//=============================================================================
// ST10_Flow5_FRobot_1.scl
// 1:1 CONVERSION FROM TIA PORTAL V18 GRAPH XML
// Generated: 2026-02-02
//=============================================================================

TYPE
    E_STEP_ST10_Flow5_FRobot_1 : (
        STEP_ST10_Flow5_FRobot_1_Tablecode_ScanFinish := 149,
        STEP_ST10_Flow5_FRobot_1_PickPalletProcess := 250,
        STEP_ST10_Flow5_FRobot_1_WaitRobotGripStatus := 360,
        STEP_ST10_Flow5_FRobot_1_WaitRobotFinish_4 := 356,
        STEP_ST10_Flow5_FRobot_1_WaitRobotFinish_9 := 371,
        STEP_ST10_Flow5_FRobot_1_WaitRobotGripStatus_4 := 372,
        STEP_ST10_Flow5_FRobot_1_WaitRobotGripHaveStatus_2 := 348,
        STEP_ST10_Flow5_FRobot_1_Open_NG_BOX_REQUESTED_ := 111,
        STEP_ST10_Flow5_FRobot_1_RobotReady_ := 311,
        STEP_ST10_Flow5_FRobot_1_WaitRobotGripStatus_6 := 378,
        STEP_ST10_Flow5_FRobot_1_Grip1SensorError := 379,
        STEP_ST10_Flow5_FRobot_1_ScanRing := 135,
        STEP_ST10_Flow5_FRobot_1_RobotAutoCycle := 329,
        STEP_ST10_Flow5_FRobot_1_RobotTaskSelect := 333,
        STEP_ST10_Flow5_FRobot_1_WaitRobotFinish_11 := 377,
        STEP_ST10_Flow5_FRobot_1_PartOKStatus_1 := 266,
        STEP_ST10_Flow5_FRobot_1_WaitRobotReachPos4 := 318,
        STEP_ST10_Flow5_FRobot_1_Step930 := 930,
        STEP_ST10_Flow5_FRobot_1_WaitR1MaintenPosFinsh := 702,
        STEP_ST10_Flow5_FRobot_1_WaitRobotGripStatus_3 := 369,
        STEP_ST10_Flow5_FRobot_1_WaitBrakeTestFinish := 921,
        STEP_ST10_Flow5_FRobot_1_PartOKStatus := 249,
        STEP_ST10_Flow5_FRobot_1_WaitGripperPos3ScanFinish := 340,
        STEP_ST10_Flow5_FRobot_1_DataMove_2 := 257,
        STEP_ST10_Flow5_FRobot_1_PressPick := 150,
        STEP_ST10_Flow5_FRobot_1_GripStatusCheck := 330,
        STEP_ST10_Flow5_FRobot_1_DataMove_5 := 264,
        STEP_ST10_Flow5_FRobot_1_NG2_PutProcessFinish := 799,
        STEP_ST10_Flow5_FRobot_1_WaitRobotReachPos5 := 321,
        STEP_ST10_Flow5_FRobot_1_StartRobotGluePut := 367,
        STEP_ST10_Flow5_FRobot_1_NG1Put_1_Press := 160,
        STEP_ST10_Flow5_FRobot_1_F5_Initial := 1,
        STEP_ST10_Flow5_FRobot_1_BrakeTestFinish := 929,
        STEP_ST10_Flow5_FRobot_1_StartRobotNG2Put_1 := 373,
        STEP_ST10_Flow5_FRobot_1_WaitPos4ScanFinish := 319,
        STEP_ST10_Flow5_FRobot_1_WaitRobotFinish := 327,
        STEP_ST10_Flow5_FRobot_1_WaitR1HomePosFinsh_1 := 899,
        STEP_ST10_Flow5_FRobot_1_NG1Put_2_ShaftScan := 165,
        STEP_ST10_Flow5_FRobot_1_FlagReset := 383,
        STEP_ST10_Flow5_FRobot_1_PressRingPutProcessFinish := 599,
        STEP_ST10_Flow5_FRobot_1_StartRobotNG3Put := 376,
        STEP_ST10_Flow5_FRobot_1_ScanStart := 246,
        STEP_ST10_Flow5_FRobot_1_StartRobotPutBuffer := 328,
        STEP_ST10_Flow5_FRobot_1_WaitMasteringTestFinish := 911,
        STEP_ST10_Flow5_FRobot_1_WaitRobotStartHome := 381,
        STEP_ST10_Flow5_FRobot_1_WaitScanCompletely := 247,
        STEP_ST10_Flow5_FRobot_1_DataMove_4 := 262,
        STEP_ST10_Flow5_FRobot_1_Grip1PartStatus := 243,
        STEP_ST10_Flow5_FRobot_1_StartRobotScanGripperCode := 334,
        STEP_ST10_Flow5_FRobot_1_WaitRobotFinish_5 := 359,
        STEP_ST10_Flow5_FRobot_1_WaitRobotGripHaveStatus := 346,
        STEP_ST10_Flow5_FRobot_1_WaitRobotFinish_1 := 343,
        STEP_ST10_Flow5_FRobot_1_WaitGripperPos1ScanFinish := 336,
        STEP_ST10_Flow5_FRobot_1_RobotStart := 316,
        STEP_ST10_Flow5_FRobot_1_WaitRobotReachPos2 := 313,
        STEP_ST10_Flow5_FRobot_1_PressShaftPut := 140,
        STEP_ST10_Flow5_FRobot_1_RobotHome := 317,
        STEP_ST10_Flow5_FRobot_1_WaitGripperPos4ScanFinish := 342,
        STEP_ST10_Flow5_FRobot_1_WaitRobotFinish_3 := 353,
        STEP_ST10_Flow5_FRobot_1_WaitRobotGripStatus_1 := 363,
        STEP_ST10_Flow5_FRobot_1_WaitPos2ScanFinish := 312,
        STEP_ST10_Flow5_FRobot_1_S10_InitialFinish := 10,
        STEP_ST10_Flow5_FRobot_1_PutBufferFinish_1 := 349,
        STEP_ST10_Flow5_FRobot_1_WaitRobotFinish_6 := 362,
        STEP_ST10_Flow5_FRobot_1_RobotScanGripperReachPos2 := 337,
        STEP_ST10_Flow5_FRobot_1_Grip2PartStatus := 244,
        STEP_ST10_Flow5_FRobot_1_WaitRobotGripStatus_2 := 366,
        STEP_ST10_Flow5_FRobot_1_WaitRobotReachPos6 := 322,
        STEP_ST10_Flow5_FRobot_1_RobotSpeed := 4,
        STEP_ST10_Flow5_FRobot_1_RobotTest := 900,
        STEP_ST10_Flow5_FRobot_1_WaitRobotHomeRequest := 703,
        STEP_ST10_Flow5_FRobot_1_PutBuffer := 120,
        STEP_ST10_Flow5_FRobot_1_StartRobotPickTable := 352,
        STEP_ST10_Flow5_FRobot_1_PickBufferFinish := 399,
        STEP_ST10_Flow5_FRobot_1_RobotScanGripperReachPos3 := 339,
        STEP_ST10_Flow5_FRobot_1_Grip2SensorError := 380,
        STEP_ST10_Flow5_FRobot_1_StartRobotPressPick := 364,
        STEP_ST10_Flow5_FRobot_1_ScanRingProcess := 450,
        STEP_ST10_Flow5_FRobot_1_GluePutProcess := 650,
        STEP_ST10_Flow5_FRobot_1_NG_2_PutProcess := 750,
        STEP_ST10_Flow5_FRobot_1_StartRobotNGPut := 370,
        STEP_ST10_Flow5_FRobot_1_Data_Clear_2 := 258,
        STEP_ST10_Flow5_FRobot_1_DataClear := 252,
        STEP_ST10_Flow5_FRobot_1_PressPickProcessFinish_ := 649,
        STEP_ST10_Flow5_FRobot_1_PickBuffer := 125,
        STEP_ST10_Flow5_FRobot_1_PickTableProcessFinish := 449,
        STEP_ST10_Flow5_FRobot_1_PressRingPutProcess := 550,
        STEP_ST10_Flow5_FRobot_1_NG_PutProcess := 700,
        STEP_ST10_Flow5_FRobot_1_WaitRobotFinish_2 := 345,
        STEP_ST10_Flow5_FRobot_1_PressRingPut := 145,
        STEP_ST10_Flow5_FRobot_1_WaitRobotGripHaveStatus_3 := 354,
        STEP_ST10_Flow5_FRobot_1_PickTableProcess := 400,
        STEP_ST10_Flow5_FRobot_1_WaitRobotReachPos3 := 314,
        STEP_ST10_Flow5_FRobot_1_Maintenance_Pos := 850,
        STEP_ST10_Flow5_FRobot_1_PressPickProcess := 600,
        STEP_ST10_Flow5_FRobot_1_Data_Clear_9 := 269,
        STEP_ST10_Flow5_FRobot_1_ProcessStart := 100,
        STEP_ST10_Flow5_FRobot_1_WaitGripperPos2ScanFinish := 338,
        STEP_ST10_Flow5_FRobot_1_Gripe2StatusAlarm := 332,
        STEP_ST10_Flow5_FRobot_1_MasteringTest_Req := 910,
        STEP_ST10_Flow5_FRobot_1_Tablecode_Scan := 200,
        STEP_ST10_Flow5_FRobot_1_Data_Clear_8 := 268,
        STEP_ST10_Flow5_FRobot_1_MES_Online__offline_ := 384,
        STEP_ST10_Flow5_FRobot_1_PartNGStatus := 251,
        STEP_ST10_Flow5_FRobot_1_S5_MESInitial := 5,
        STEP_ST10_Flow5_FRobot_1_StartRobotScanFixtureCode := 308,
        STEP_ST10_Flow5_FRobot_1_BrakeTest_Req := 920,
        STEP_ST10_Flow5_FRobot_1_WaitPos5ScanFinish := 320,
        STEP_ST10_Flow5_FRobot_1_RobotScanGripperReachPos4 := 341,
        STEP_ST10_Flow5_FRobot_1_ScanRingProcessFinish := 499,
        STEP_ST10_Flow5_FRobot_1_WaitRobotGripStatus_5 := 375,
        STEP_ST10_Flow5_FRobot_1_Masref_test := 132,
        STEP_ST10_Flow5_FRobot_1_WaitPos1ScanFinish := 310,
        STEP_ST10_Flow5_FRobot_1_StartRobotPressShaftPut := 358,
        STEP_ST10_Flow5_FRobot_1_StartRobotPickBuffer := 344,
        STEP_ST10_Flow5_FRobot_1_PressShaftPutProcess := 500,
        STEP_ST10_Flow5_FRobot_1_StartRobotPressRingPut := 361,
        STEP_ST10_Flow5_FRobot_1_NG1Put_3_RingScan := 170,
        STEP_ST10_Flow5_FRobot_1_NG1_PutProcessFinish := 749,
        STEP_ST10_Flow5_FRobot_1_WaitRobotReachScanPos := 357,
        STEP_ST10_Flow5_FRobot_1_PickPallet := 115,
        STEP_ST10_Flow5_FRobot_1_ScanFixtureCode := 110,
        STEP_ST10_Flow5_FRobot_1_PutBufferProcess := 300,
        STEP_ST10_Flow5_FRobot_1_WaitRobotFinish_10 := 374,
        STEP_ST10_Flow5_FRobot_1_ReqRobotToHomePos := 704,
        STEP_ST10_Flow5_FRobot_1_DataMove_1 := 255,
        STEP_ST10_Flow5_FRobot_1_Maintenance := 131,
        STEP_ST10_Flow5_FRobot_1_GluePut := 155,
        STEP_ST10_Flow5_FRobot_1_PickBufferProcess := 350,
        STEP_ST10_Flow5_FRobot_1_GluePutProcessFinish := 699,
        STEP_ST10_Flow5_FRobot_1_PickPalletFinish := 299,
        STEP_ST10_Flow5_FRobot_1_DataMove := 253,
        STEP_ST10_Flow5_FRobot_1_PressShaftPutProcessFinish := 549,
        STEP_ST10_Flow5_FRobot_1_StartRobotScanRing := 355,
        STEP_ST10_Flow5_FRobot_1_RobotManuallyMoved_ := 382,
        STEP_ST10_Flow5_FRobot_1_RobotScanGripperReachPos1 := 335,
        STEP_ST10_Flow5_FRobot_1_Data_Clear_7 := 267,
        STEP_ST10_Flow5_FRobot_1_CheckScanReady := 245,
        STEP_ST10_Flow5_FRobot_1_Brake_Test := 133,
        STEP_ST10_Flow5_FRobot_1_ReqRobotToMantenPos := 701,
        STEP_ST10_Flow5_FRobot_1_NG3_PutProcessFinish := 849,
        STEP_ST10_Flow5_FRobot_1_NG_3_PutProcess := 800,
        STEP_ST10_Flow5_FRobot_1_Wait_ScanFinish := 242,
        STEP_ST10_Flow5_FRobot_1_WaitRobotReachPos1 := 309,
        STEP_ST10_Flow5_FRobot_1_WaitRobotGripHaveStatus_1 := 347,
        STEP_ST10_Flow5_FRobot_1_DataMove_3 := 260,
        STEP_ST10_Flow5_FRobot_1_MasteringTestFinish := 919,
        STEP_ST10_Flow5_FRobot_1_StartRobotPickPalletShaft := 326,
        STEP_ST10_Flow5_FRobot_1_PickTable := 130,
        STEP_ST10_Flow5_FRobot_1_WaitRobotFinish_8 := 368,
        STEP_ST10_Flow5_FRobot_1_Gripe1StatusAlarm := 331,
        STEP_ST10_Flow5_FRobot_1_CodeMove := 248,
        STEP_ST10_Flow5_FRobot_1_WaitPos3ScanFinish := 315,
        STEP_ST10_Flow5_FRobot_1_WaitRobotFinish_7 := 365,
    ) INT := 1;
END_TYPE

CONST
    STEP_ST10_Flow5_FRobot_1_Tablecode_ScanFinish := 149;
    STEP_ST10_Flow5_FRobot_1_PickPalletProcess := 250;
    STEP_ST10_Flow5_FRobot_1_WaitRobotGripStatus := 360;
    STEP_ST10_Flow5_FRobot_1_WaitRobotFinish_4 := 356;
    STEP_ST10_Flow5_FRobot_1_WaitRobotFinish_9 := 371;
    STEP_ST10_Flow5_FRobot_1_WaitRobotGripStatus_4 := 372;
    STEP_ST10_Flow5_FRobot_1_WaitRobotGripHaveStatus_2 := 348;
    STEP_ST10_Flow5_FRobot_1_Open_NG_BOX_REQUESTED_ := 111;
    STEP_ST10_Flow5_FRobot_1_RobotReady_ := 311;
    STEP_ST10_Flow5_FRobot_1_WaitRobotGripStatus_6 := 378;
    STEP_ST10_Flow5_FRobot_1_Grip1SensorError := 379;
    STEP_ST10_Flow5_FRobot_1_ScanRing := 135;
    STEP_ST10_Flow5_FRobot_1_RobotAutoCycle := 329;
    STEP_ST10_Flow5_FRobot_1_RobotTaskSelect := 333;
    STEP_ST10_Flow5_FRobot_1_WaitRobotFinish_11 := 377;
    STEP_ST10_Flow5_FRobot_1_PartOKStatus_1 := 266;
    STEP_ST10_Flow5_FRobot_1_WaitRobotReachPos4 := 318;
    STEP_ST10_Flow5_FRobot_1_Step930 := 930;
    STEP_ST10_Flow5_FRobot_1_WaitR1MaintenPosFinsh := 702;
    STEP_ST10_Flow5_FRobot_1_WaitRobotGripStatus_3 := 369;
    STEP_ST10_Flow5_FRobot_1_WaitBrakeTestFinish := 921;
    STEP_ST10_Flow5_FRobot_1_PartOKStatus := 249;
    STEP_ST10_Flow5_FRobot_1_WaitGripperPos3ScanFinish := 340;
    STEP_ST10_Flow5_FRobot_1_DataMove_2 := 257;
    STEP_ST10_Flow5_FRobot_1_PressPick := 150;
    STEP_ST10_Flow5_FRobot_1_GripStatusCheck := 330;
    STEP_ST10_Flow5_FRobot_1_DataMove_5 := 264;
    STEP_ST10_Flow5_FRobot_1_NG2_PutProcessFinish := 799;
    STEP_ST10_Flow5_FRobot_1_WaitRobotReachPos5 := 321;
    STEP_ST10_Flow5_FRobot_1_StartRobotGluePut := 367;
    STEP_ST10_Flow5_FRobot_1_NG1Put_1_Press := 160;
    STEP_ST10_Flow5_FRobot_1_F5_Initial := 1;
    STEP_ST10_Flow5_FRobot_1_BrakeTestFinish := 929;
    STEP_ST10_Flow5_FRobot_1_StartRobotNG2Put_1 := 373;
    STEP_ST10_Flow5_FRobot_1_WaitPos4ScanFinish := 319;
    STEP_ST10_Flow5_FRobot_1_WaitRobotFinish := 327;
    STEP_ST10_Flow5_FRobot_1_WaitR1HomePosFinsh_1 := 899;
    STEP_ST10_Flow5_FRobot_1_NG1Put_2_ShaftScan := 165;
    STEP_ST10_Flow5_FRobot_1_FlagReset := 383;
    STEP_ST10_Flow5_FRobot_1_PressRingPutProcessFinish := 599;
    STEP_ST10_Flow5_FRobot_1_StartRobotNG3Put := 376;
    STEP_ST10_Flow5_FRobot_1_ScanStart := 246;
    STEP_ST10_Flow5_FRobot_1_StartRobotPutBuffer := 328;
    STEP_ST10_Flow5_FRobot_1_WaitMasteringTestFinish := 911;
    STEP_ST10_Flow5_FRobot_1_WaitRobotStartHome := 381;
    STEP_ST10_Flow5_FRobot_1_WaitScanCompletely := 247;
    STEP_ST10_Flow5_FRobot_1_DataMove_4 := 262;
    STEP_ST10_Flow5_FRobot_1_Grip1PartStatus := 243;
    STEP_ST10_Flow5_FRobot_1_StartRobotScanGripperCode := 334;
    STEP_ST10_Flow5_FRobot_1_WaitRobotFinish_5 := 359;
    STEP_ST10_Flow5_FRobot_1_WaitRobotGripHaveStatus := 346;
    STEP_ST10_Flow5_FRobot_1_WaitRobotFinish_1 := 343;
    STEP_ST10_Flow5_FRobot_1_WaitGripperPos1ScanFinish := 336;
    STEP_ST10_Flow5_FRobot_1_RobotStart := 316;
    STEP_ST10_Flow5_FRobot_1_WaitRobotReachPos2 := 313;
    STEP_ST10_Flow5_FRobot_1_PressShaftPut := 140;
    STEP_ST10_Flow5_FRobot_1_RobotHome := 317;
    STEP_ST10_Flow5_FRobot_1_WaitGripperPos4ScanFinish := 342;
    STEP_ST10_Flow5_FRobot_1_WaitRobotFinish_3 := 353;
    STEP_ST10_Flow5_FRobot_1_WaitRobotGripStatus_1 := 363;
    STEP_ST10_Flow5_FRobot_1_WaitPos2ScanFinish := 312;
    STEP_ST10_Flow5_FRobot_1_S10_InitialFinish := 10;
    STEP_ST10_Flow5_FRobot_1_PutBufferFinish_1 := 349;
    STEP_ST10_Flow5_FRobot_1_WaitRobotFinish_6 := 362;
    STEP_ST10_Flow5_FRobot_1_RobotScanGripperReachPos2 := 337;
    STEP_ST10_Flow5_FRobot_1_Grip2PartStatus := 244;
    STEP_ST10_Flow5_FRobot_1_WaitRobotGripStatus_2 := 366;
    STEP_ST10_Flow5_FRobot_1_WaitRobotReachPos6 := 322;
    STEP_ST10_Flow5_FRobot_1_RobotSpeed := 4;
    STEP_ST10_Flow5_FRobot_1_RobotTest := 900;
    STEP_ST10_Flow5_FRobot_1_WaitRobotHomeRequest := 703;
    STEP_ST10_Flow5_FRobot_1_PutBuffer := 120;
    STEP_ST10_Flow5_FRobot_1_StartRobotPickTable := 352;
    STEP_ST10_Flow5_FRobot_1_PickBufferFinish := 399;
    STEP_ST10_Flow5_FRobot_1_RobotScanGripperReachPos3 := 339;
    STEP_ST10_Flow5_FRobot_1_Grip2SensorError := 380;
    STEP_ST10_Flow5_FRobot_1_StartRobotPressPick := 364;
    STEP_ST10_Flow5_FRobot_1_ScanRingProcess := 450;
    STEP_ST10_Flow5_FRobot_1_GluePutProcess := 650;
    STEP_ST10_Flow5_FRobot_1_NG_2_PutProcess := 750;
    STEP_ST10_Flow5_FRobot_1_StartRobotNGPut := 370;
    STEP_ST10_Flow5_FRobot_1_Data_Clear_2 := 258;
    STEP_ST10_Flow5_FRobot_1_DataClear := 252;
    STEP_ST10_Flow5_FRobot_1_PressPickProcessFinish_ := 649;
    STEP_ST10_Flow5_FRobot_1_PickBuffer := 125;
    STEP_ST10_Flow5_FRobot_1_PickTableProcessFinish := 449;
    STEP_ST10_Flow5_FRobot_1_PressRingPutProcess := 550;
    STEP_ST10_Flow5_FRobot_1_NG_PutProcess := 700;
    STEP_ST10_Flow5_FRobot_1_WaitRobotFinish_2 := 345;
    STEP_ST10_Flow5_FRobot_1_PressRingPut := 145;
    STEP_ST10_Flow5_FRobot_1_WaitRobotGripHaveStatus_3 := 354;
    STEP_ST10_Flow5_FRobot_1_PickTableProcess := 400;
    STEP_ST10_Flow5_FRobot_1_WaitRobotReachPos3 := 314;
    STEP_ST10_Flow5_FRobot_1_Maintenance_Pos := 850;
    STEP_ST10_Flow5_FRobot_1_PressPickProcess := 600;
    STEP_ST10_Flow5_FRobot_1_Data_Clear_9 := 269;
    STEP_ST10_Flow5_FRobot_1_ProcessStart := 100;
    STEP_ST10_Flow5_FRobot_1_WaitGripperPos2ScanFinish := 338;
    STEP_ST10_Flow5_FRobot_1_Gripe2StatusAlarm := 332;
    STEP_ST10_Flow5_FRobot_1_MasteringTest_Req := 910;
    STEP_ST10_Flow5_FRobot_1_Tablecode_Scan := 200;
    STEP_ST10_Flow5_FRobot_1_Data_Clear_8 := 268;
    STEP_ST10_Flow5_FRobot_1_MES_Online__offline_ := 384;
    STEP_ST10_Flow5_FRobot_1_PartNGStatus := 251;
    STEP_ST10_Flow5_FRobot_1_S5_MESInitial := 5;
    STEP_ST10_Flow5_FRobot_1_StartRobotScanFixtureCode := 308;
    STEP_ST10_Flow5_FRobot_1_BrakeTest_Req := 920;
    STEP_ST10_Flow5_FRobot_1_WaitPos5ScanFinish := 320;
    STEP_ST10_Flow5_FRobot_1_RobotScanGripperReachPos4 := 341;
    STEP_ST10_Flow5_FRobot_1_ScanRingProcessFinish := 499;
    STEP_ST10_Flow5_FRobot_1_WaitRobotGripStatus_5 := 375;
    STEP_ST10_Flow5_FRobot_1_Masref_test := 132;
    STEP_ST10_Flow5_FRobot_1_WaitPos1ScanFinish := 310;
    STEP_ST10_Flow5_FRobot_1_StartRobotPressShaftPut := 358;
    STEP_ST10_Flow5_FRobot_1_StartRobotPickBuffer := 344;
    STEP_ST10_Flow5_FRobot_1_PressShaftPutProcess := 500;
    STEP_ST10_Flow5_FRobot_1_StartRobotPressRingPut := 361;
    STEP_ST10_Flow5_FRobot_1_NG1Put_3_RingScan := 170;
    STEP_ST10_Flow5_FRobot_1_NG1_PutProcessFinish := 749;
    STEP_ST10_Flow5_FRobot_1_WaitRobotReachScanPos := 357;
    STEP_ST10_Flow5_FRobot_1_PickPallet := 115;
    STEP_ST10_Flow5_FRobot_1_ScanFixtureCode := 110;
    STEP_ST10_Flow5_FRobot_1_PutBufferProcess := 300;
    STEP_ST10_Flow5_FRobot_1_WaitRobotFinish_10 := 374;
    STEP_ST10_Flow5_FRobot_1_ReqRobotToHomePos := 704;
    STEP_ST10_Flow5_FRobot_1_DataMove_1 := 255;
    STEP_ST10_Flow5_FRobot_1_Maintenance := 131;
    STEP_ST10_Flow5_FRobot_1_GluePut := 155;
    STEP_ST10_Flow5_FRobot_1_PickBufferProcess := 350;
    STEP_ST10_Flow5_FRobot_1_GluePutProcessFinish := 699;
    STEP_ST10_Flow5_FRobot_1_PickPalletFinish := 299;
    STEP_ST10_Flow5_FRobot_1_DataMove := 253;
    STEP_ST10_Flow5_FRobot_1_PressShaftPutProcessFinish := 549;
    STEP_ST10_Flow5_FRobot_1_StartRobotScanRing := 355;
    STEP_ST10_Flow5_FRobot_1_RobotManuallyMoved_ := 382;
    STEP_ST10_Flow5_FRobot_1_RobotScanGripperReachPos1 := 335;
    STEP_ST10_Flow5_FRobot_1_Data_Clear_7 := 267;
    STEP_ST10_Flow5_FRobot_1_CheckScanReady := 245;
    STEP_ST10_Flow5_FRobot_1_Brake_Test := 133;
    STEP_ST10_Flow5_FRobot_1_ReqRobotToMantenPos := 701;
    STEP_ST10_Flow5_FRobot_1_NG3_PutProcessFinish := 849;
    STEP_ST10_Flow5_FRobot_1_NG_3_PutProcess := 800;
    STEP_ST10_Flow5_FRobot_1_Wait_ScanFinish := 242;
    STEP_ST10_Flow5_FRobot_1_WaitRobotReachPos1 := 309;
    STEP_ST10_Flow5_FRobot_1_WaitRobotGripHaveStatus_1 := 347;
    STEP_ST10_Flow5_FRobot_1_DataMove_3 := 260;
    STEP_ST10_Flow5_FRobot_1_MasteringTestFinish := 919;
    STEP_ST10_Flow5_FRobot_1_StartRobotPickPalletShaft := 326;
    STEP_ST10_Flow5_FRobot_1_PickTable := 130;
    STEP_ST10_Flow5_FRobot_1_WaitRobotFinish_8 := 368;
    STEP_ST10_Flow5_FRobot_1_Gripe1StatusAlarm := 331;
    STEP_ST10_Flow5_FRobot_1_CodeMove := 248;
    STEP_ST10_Flow5_FRobot_1_WaitPos3ScanFinish := 315;
    STEP_ST10_Flow5_FRobot_1_WaitRobotFinish_7 := 365;
END_CONST

FUNCTION_BLOCK "ST10_Flow5_FRobot_1_1to1"
{ S7_Optimized_Access := 'TRUE' }
VERSION : 1.0

VAR_INPUT
    iSysInface : "RCS_SysComInterface_V1";
END_VAR

VAR_IN_OUT
    ioPM_Inface : "RCS_PMInterface_V1";
    ioStatus : Int;
END_VAR

VAR_OUTPUT
    oAlarmID : Int;
END_VAR

VAR
    State : INT := 1;
    act_InitialRun : Bool;
    act_InitialOK : Bool;
    act_WaitRunning : Bool;
    act_Running : Bool;
    act_ProcessComplete : Bool;
    act_ProcessStart : Bool;
    act_UnPause : Bool;
    bError : Bool;
    wErrorID : Word;
END_VAR

BEGIN
    //======================================================================
    // STATE MACHINE - Inline Transition Conditions
    //======================================================================

    CASE #State OF

        // ===========================================
        // STEP 149: Tablecode ScanFinish
        // ===========================================
        STEP_ST10_Flow5_FRobot_1_Tablecode_ScanFinish:
            // Action Qualifier=S
            // Token: #ioPM_Inface.ProcessComplete
            #ioPM_Inface.ProcessComplete := TRUE;
            // Action Qualifier=R
            // Token: #ioPM_Inface.ProcessStart
            #ioPM_Inface.ProcessStart := FALSE;

            // Transition to next step: 250
            IF TRUE THEN  // Sequential transition - review XML for actual condition
                #State := STEP_ST10_Flow5_FRobot_1_PickPalletProcess;
            END_IF;

        // ===========================================
        // STEP 250: PickPalletProcess
        // ===========================================
        STEP_ST10_Flow5_FRobot_1_PickPalletProcess:
            // No actions in XML

            // Transition to next step: 360
            IF TRUE THEN  // Sequential transition - review XML for actual condition
                #State := STEP_ST10_Flow5_FRobot_1_WaitRobotGripStatus;
            END_IF;

        // ===========================================
        // STEP 360: WaitRobotGripStatus
        // ===========================================
        STEP_ST10_Flow5_FRobot_1_WaitRobotGripStatus:
            // No actions in XML

            // Transition to next step: 356
            IF TRUE THEN  // Sequential transition - review XML for actual condition
                #State := STEP_ST10_Flow5_FRobot_1_WaitRobotFinish_4;
            END_IF;

        // ===========================================
        // STEP 356: WaitRobotFinish_4
        // ===========================================
        STEP_ST10_Flow5_FRobot_1_WaitRobotFinish_4:
            // Action Qualifier=N
            // Token: "KukaRobot1_CtrlDB".sPLCtoROB.User.Cycle.DI262_RingScanComplete
            "KukaRobot1_CtrlDB".sPLCtoROB.User.Cycle.DI262_RingScanComplete;

            // Transition to next step: 371
            IF TRUE THEN  // Sequential transition - review XML for actual condition
                #State := STEP_ST10_Flow5_FRobot_1_WaitRobotFinish_9;
            END_IF;

        // ===========================================
        // STEP 371: WaitRobotFinish_9
        // ===========================================
        STEP_ST10_Flow5_FRobot_1_WaitRobotFinish_9:
            // No actions in XML

            // Transition to next step: 372
            IF TRUE THEN  // Sequential transition - review XML for actual condition
                #State := STEP_ST10_Flow5_FRobot_1_WaitRobotGripStatus_4;
            END_IF;

        // ===========================================
        // STEP 372: WaitRobotGripStatus_4
        // ===========================================
        STEP_ST10_Flow5_FRobot_1_WaitRobotGripStatus_4:
            // No actions in XML

            // Transition to next step: 348
            IF TRUE THEN  // Sequential transition - review XML for actual condition
                #State := STEP_ST10_Flow5_FRobot_1_WaitRobotGripHaveStatus_2;
            END_IF;

        // ===========================================
        // STEP 348: WaitRobotGripHaveStatus_2
        // ===========================================
        STEP_ST10_Flow5_FRobot_1_WaitRobotGripHaveStatus_2:
            // No actions in XML

            // Transition to next step: 111
            IF TRUE THEN  // Sequential transition - review XML for actual condition
                #State := STEP_ST10_Flow5_FRobot_1_Open_NG_BOX_REQUESTED_;
            END_IF;

        // ===========================================
        // STEP 111: Open NG BOX REQUESTED?
        // ===========================================
        STEP_ST10_Flow5_FRobot_1_Open_NG_BOX_REQUESTED_:
            // No actions in XML

            // Transition to next step: 311
            IF TRUE THEN  // Sequential transition - review XML for actual condition
                #State := STEP_ST10_Flow5_FRobot_1_RobotReady_;
            END_IF;

        // ===========================================
        // STEP 311: RobotReady?
        // ===========================================
        STEP_ST10_Flow5_FRobot_1_RobotReady_:
            // No actions in XML

            // Transition to next step: 378
            IF TRUE THEN  // Sequential transition - review XML for actual condition
                #State := STEP_ST10_Flow5_FRobot_1_WaitRobotGripStatus_6;
            END_IF;

        // ===========================================
        // STEP 378: WaitRobotGripStatus_6
        // ===========================================
        STEP_ST10_Flow5_FRobot_1_WaitRobotGripStatus_6:
            // No actions in XML

            // Transition to next step: 379
            IF TRUE THEN  // Sequential transition - review XML for actual condition
                #State := STEP_ST10_Flow5_FRobot_1_Grip1SensorError;
            END_IF;

        // ===========================================
        // STEP 379: Grip1SensorError
        // ===========================================
        STEP_ST10_Flow5_FRobot_1_Grip1SensorError:
            // No actions in XML

            // Transition to next step: 135
            IF TRUE THEN  // Sequential transition - review XML for actual condition
                #State := STEP_ST10_Flow5_FRobot_1_ScanRing;
            END_IF;

        // ===========================================
        // STEP 135: ScanRing
        // ===========================================
        STEP_ST10_Flow5_FRobot_1_ScanRing:
            // Action Qualifier=R
            // Token: #ioPM_Inface.ProcessComplete
            #ioPM_Inface.ProcessComplete := FALSE;
            // Action Qualifier=S
            // Token: #ioPM_Inface.ProcessStart
            #ioPM_Inface.ProcessStart := TRUE;

            // Transition to next step: 329
            IF TRUE THEN  // Sequential transition - review XML for actual condition
                #State := STEP_ST10_Flow5_FRobot_1_RobotAutoCycle;
            END_IF;

        // ===========================================
        // STEP 329: RobotAutoCycle
        // ===========================================
        STEP_ST10_Flow5_FRobot_1_RobotAutoCycle:
            // Action Qualifier=N
            // Token: "KukaRobot1_CtrlDB".ioStartAutoCycle
            "KukaRobot1_CtrlDB".ioStartAutoCycle;

            // Transition to next step: 333
            IF TRUE THEN  // Sequential transition - review XML for actual condition
                #State := STEP_ST10_Flow5_FRobot_1_RobotTaskSelect;
            END_IF;

        // ===========================================
        // STEP 333: RobotTaskSelect
        // ===========================================
        STEP_ST10_Flow5_FRobot_1_RobotTaskSelect:
            // No actions in XML

            // Transition to next step: 377
            IF TRUE THEN  // Sequential transition - review XML for actual condition
                #State := STEP_ST10_Flow5_FRobot_1_WaitRobotFinish_11;
            END_IF;

        // ===========================================
        // STEP 377: WaitRobotFinish_11
        // ===========================================
        STEP_ST10_Flow5_FRobot_1_WaitRobotFinish_11:
            // No actions in XML

            // Transition to next step: 266
            IF TRUE THEN  // Sequential transition - review XML for actual condition
                #State := STEP_ST10_Flow5_FRobot_1_PartOKStatus_1;
            END_IF;

        // ===========================================
        // STEP 266: PartOKStatus_1
        // ===========================================
        STEP_ST10_Flow5_FRobot_1_PartOKStatus_1:
            // Action Qualifier=N
            // Token: "AutoProcessData".F_Robot1Grip2.PartStatus := 110
            "AutoProcessData".F_Robot1Grip2.PartStatus := 110;

            // Transition to next step: 318
            IF TRUE THEN  // Sequential transition - review XML for actual condition
                #State := STEP_ST10_Flow5_FRobot_1_WaitRobotReachPos4;
            END_IF;

        // ===========================================
        // STEP 318: WaitRobotReachPos4
        // ===========================================
        STEP_ST10_Flow5_FRobot_1_WaitRobotReachPos4:
            // No actions in XML

            // Transition to next step: 930
            IF TRUE THEN  // Sequential transition - review XML for actual condition
                #State := STEP_ST10_Flow5_FRobot_1_Step930;
            END_IF;

        // ===========================================
        // STEP 930: Step930
        // ===========================================
        STEP_ST10_Flow5_FRobot_1_Step930:
            // No actions in XML

            // Transition to next step: 702
            IF TRUE THEN  // Sequential transition - review XML for actual condition
                #State := STEP_ST10_Flow5_FRobot_1_WaitR1MaintenPosFinsh;
            END_IF;

        // ===========================================
        // STEP 702: WaitR1MaintenPosFinsh
        // ===========================================
        STEP_ST10_Flow5_FRobot_1_WaitR1MaintenPosFinsh:
            // Action Qualifier=R
            // Token: "AutoProcessControl".Robot_1.MaintenanceRequest
            "AutoProcessControl".Robot_1.MaintenanceRequest := FALSE;

            // Transition to next step: 369
            IF TRUE THEN  // Sequential transition - review XML for actual condition
                #State := STEP_ST10_Flow5_FRobot_1_WaitRobotGripStatus_3;
            END_IF;

        // ===========================================
        // STEP 369: WaitRobotGripStatus_3
        // ===========================================
        STEP_ST10_Flow5_FRobot_1_WaitRobotGripStatus_3:
            // No actions in XML

            // Transition to next step: 921
            IF TRUE THEN  // Sequential transition - review XML for actual condition
                #State := STEP_ST10_Flow5_FRobot_1_WaitBrakeTestFinish;
            END_IF;

        // ===========================================
        // STEP 921: WaitBrakeTestFinish
        // ===========================================
        STEP_ST10_Flow5_FRobot_1_WaitBrakeTestFinish:
            // No actions in XML

            // Transition to next step: 249
            IF TRUE THEN  // Sequential transition - review XML for actual condition
                #State := STEP_ST10_Flow5_FRobot_1_PartOKStatus;
            END_IF;

        // ===========================================
        // STEP 249: PartOKStatus
        // ===========================================
        STEP_ST10_Flow5_FRobot_1_PartOKStatus:
            // Action Qualifier=N
            // Token: "AutoProcessData".F_Robot1Grip2.PartStatus := 199
            "AutoProcessData".F_Robot1Grip2.PartStatus := 199;

            // Transition to next step: 340
            IF TRUE THEN  // Sequential transition - review XML for actual condition
                #State := STEP_ST10_Flow5_FRobot_1_WaitGripperPos3ScanFinish;
            END_IF;

        // ===========================================
        // STEP 340: WaitGripperPos3ScanFinish
        // ===========================================
        STEP_ST10_Flow5_FRobot_1_WaitGripperPos3ScanFinish:
            // No actions in XML

            // Transition to next step: 257
            IF TRUE THEN  // Sequential transition - review XML for actual condition
                #State := STEP_ST10_Flow5_FRobot_1_DataMove_2;
            END_IF;

        // ===========================================
        // STEP 257: DataMove_2
        // ===========================================
        STEP_ST10_Flow5_FRobot_1_DataMove_2:
            // Action Qualifier=N, Event="S1"
            // Token: "AutoProcessData".B_Press1 := "AutoProcessData".F_Robot1Grip1
            "AutoProcessData".B_Press1 := "AutoProcessData".F_Robot1Grip1;
            // Action Qualifier=N, Event="S1"
            // Token: "AutoProcessData".F_Robot1Grip1 := "AutoProcessData".ClearData
            "AutoProcessData".F_Robot1Grip1 := "AutoProcessData".ClearData;

            // Transition to next step: 150
            IF TRUE THEN  // Sequential transition - review XML for actual condition
                #State := STEP_ST10_Flow5_FRobot_1_PressPick;
            END_IF;

        // ===========================================
        // STEP 150: PressPick
        // ===========================================
        STEP_ST10_Flow5_FRobot_1_PressPick:
            // Action Qualifier=R
            // Token: #ioPM_Inface.ProcessComplete
            #ioPM_Inface.ProcessComplete := FALSE;
            // Action Qualifier=S
            // Token: #ioPM_Inface.ProcessStart
            #ioPM_Inface.ProcessStart := TRUE;

            // Transition to next step: 330
            IF TRUE THEN  // Sequential transition - review XML for actual condition
                #State := STEP_ST10_Flow5_FRobot_1_GripStatusCheck;
            END_IF;

        // ===========================================
        // STEP 330: GripStatusCheck
        // ===========================================
        STEP_ST10_Flow5_FRobot_1_GripStatusCheck:
            // No actions in XML

            // Transition to next step: 264
            IF TRUE THEN  // Sequential transition - review XML for actual condition
                #State := STEP_ST10_Flow5_FRobot_1_DataMove_5;
            END_IF;

        // ===========================================
        // STEP 264: DataMove_5
        // ===========================================
        STEP_ST10_Flow5_FRobot_1_DataMove_5:
            // Action Qualifier=N, Event="S1"
            // Token: "AutoProcessData".C_Glue := "AutoProcessData".F_Robot1Grip1
            "AutoProcessData".C_Glue := "AutoProcessData".F_Robot1Grip1;
            // Action Qualifier=N, Event="S1"
            // Token: "AutoProcessData".F_Robot1Grip1 := "AutoProcessData".ClearData
            "AutoProcessData".F_Robot1Grip1 := "AutoProcessData".ClearData;

            // Transition to next step: 799
            IF TRUE THEN  // Sequential transition - review XML for actual condition
                #State := STEP_ST10_Flow5_FRobot_1_NG2_PutProcessFinish;
            END_IF;

        // ===========================================
        // STEP 799: NG2 PutProcessFinish
        // ===========================================
        STEP_ST10_Flow5_FRobot_1_NG2_PutProcessFinish:
            // Action Qualifier=S
            // Token: #ioPM_Inface.ProcessComplete
            #ioPM_Inface.ProcessComplete := TRUE;
            // Action Qualifier=R
            // Token: #ioPM_Inface.ProcessStart
            #ioPM_Inface.ProcessStart := FALSE;

            // Transition to next step: 321
            IF TRUE THEN  // Sequential transition - review XML for actual condition
                #State := STEP_ST10_Flow5_FRobot_1_WaitRobotReachPos5;
            END_IF;

        // ===========================================
        // STEP 321: WaitRobotReachPos5
        // ===========================================
        STEP_ST10_Flow5_FRobot_1_WaitRobotReachPos5:
            // No actions in XML

            // Transition to next step: 367
            IF TRUE THEN  // Sequential transition - review XML for actual condition
                #State := STEP_ST10_Flow5_FRobot_1_StartRobotGluePut;
            END_IF;

        // ===========================================
        // STEP 367: StartRobotGluePut
        // ===========================================
        STEP_ST10_Flow5_FRobot_1_StartRobotGluePut:
            // Action Qualifier=N
            // Token: "KukaRobot1_CtrlDB".sPLCtoROB.User.Cycle.DI289_GluePutReq
            "KukaRobot1_CtrlDB".sPLCtoROB.User.Cycle.DI289_GluePutReq;

            // Transition to next step: 160
            IF TRUE THEN  // Sequential transition - review XML for actual condition
                #State := STEP_ST10_Flow5_FRobot_1_NG1Put_1_Press;
            END_IF;

        // ===========================================
        // STEP 160: NG1Put_1/Press
        // ===========================================
        STEP_ST10_Flow5_FRobot_1_NG1Put_1_Press:
            // Action Qualifier=S
            // Token: "AutoProcessControl".Robot_1.NGPutFlag
            "AutoProcessControl".Robot_1.NGPutFlag := TRUE;
            // Action Qualifier=R
            // Token: #ioPM_Inface.ProcessComplete
            #ioPM_Inface.ProcessComplete := FALSE;
            // Action Qualifier=S
            // Token: #ioPM_Inface.ProcessStart
            #ioPM_Inface.ProcessStart := TRUE;

            // Transition to next step: 1
            IF TRUE THEN  // Sequential transition - review XML for actual condition
                #State := STEP_ST10_Flow5_FRobot_1_F5_Initial;
            END_IF;

        // ===========================================
        // STEP 1: F5_Initial
        // ===========================================
        STEP_ST10_Flow5_FRobot_1_F5_Initial:
            // Action Qualifier=S
            // Token: #ioPM_Inface.InitialRun
            #ioPM_Inface.InitialRun := TRUE;
            // Action Qualifier=R
            // Token: #ioPM_Inface.InitialOK
            #ioPM_Inface.InitialOK := FALSE;
            // Action Qualifier=R
            // Token: #ioPM_Inface.WaitRunning
            #ioPM_Inface.WaitRunning := FALSE;
            // Action Qualifier=R
            // Token: #ioPM_Inface.Running
            #ioPM_Inface.Running := FALSE;
            // Action Qualifier=R
            // Token: #ioPM_Inface.UnPause
            #ioPM_Inface.UnPause := FALSE;
            // Action Qualifier=R
            // Token: "Station_Sys".Cmd.Calibration
            "Station_Sys".Cmd.Calibration := FALSE;
            // Action Qualifier=R
            // Token: "Station_Sys".Cmd.ChangeOver
            "Station_Sys".Cmd.ChangeOver := FALSE;
            // Action Qualifier=N
            // Token: //"ST350_Sys".Cmd.DryRun
            //"ST350_Sys".Cmd.DryRun;
            // Action Qualifier=R
            // Token: "Station_Sys".Cmd.Reserve
            "Station_Sys".Cmd.Reserve := FALSE;
            // Action Qualifier=R
            // Token: "Station_Sys".Cmd.OneCycle
            "Station_Sys".Cmd.OneCycle := FALSE;
            // Action Qualifier=R
            // Token: "AutoProcessControl".Robot_1.GluePutFlag
            "AutoProcessControl".Robot_1.GluePutFlag := FALSE;
            // Action Qualifier=R
            // Token: "AutoProcessControl".Robot_1.NGPutFlag
            "AutoProcessControl".Robot_1.NGPutFlag := FALSE;
            // Action Qualifier=R
            // Token: #ioPM_Inface.ProcessComplete
            #ioPM_Inface.ProcessComplete := FALSE;
            // Action Qualifier=R
            // Token: #ioPM_Inface.ProcessStart
            #ioPM_Inface.ProcessStart := FALSE;
            // Action Qualifier=R
            // Token: "ChangeOver_DB".Robot_1.MaintenancePosReqSelFlag
            "ChangeOver_DB".Robot_1.MaintenancePosReqSelFlag := FALSE;
            // Action Qualifier=N
            // Token: //"Robot_DB".Robot_1.MasteringTest_Req
            //"Robot_DB".Robot_1.MasteringTest_Req;
            // Action Qualifier=N
            // Token: //"Robot_DB".Robot_1.BrakeTest_Req
            //"Robot_DB".Robot_1.BrakeTest_Req;
            // Action Qualifier=R
            // Token: "KukaRobot1_CtrlDB".sPLCtoROB.User.Cycle.DI281_PressPickShaftReq
            "KukaRobot1_CtrlDB".sPLCtoROB.User.Cycle.DI281_PressPickShaftReq := FALSE;
            // Action Qualifier=R
            // Token: "KukaRobot1_CtrlDB".sPLCtoROB.User.Cycle.DI277_PressRingPutReq
            "KukaRobot1_CtrlDB".sPLCtoROB.User.Cycle.DI277_PressRingPutReq := FALSE;
            // Action Qualifier=R
            // Token: "KukaRobot1_CtrlDB".sPLCtoROB.User.Cycle.DI278_PressRingPutLeave
            "KukaRobot1_CtrlDB".sPLCtoROB.User.Cycle.DI278_PressRingPutLeave := FALSE;
            // Action Qualifier=R
            // Token: "KukaRobot1_CtrlDB".sPLCtoROB.User.Cycle.DI267_LoadRingScanNGReq3
            "KukaRobot1_CtrlDB".sPLCtoROB.User.Cycle.DI267_LoadRingScanNGReq3 := FALSE;
            // Action Qualifier=R
            // Token: "KukaRobot1_CtrlDB".sPLCtoROB.User.Cycle.DI265_LoadPressNGReq1
            "KukaRobot1_CtrlDB".sPLCtoROB.User.Cycle.DI265_LoadPressNGReq1 := FALSE;
            // Action Qualifier=R
            // Token: "KukaRobot1_CtrlDB".sPLCtoROB.User.Cycle.DI261_RingScanReq
            "KukaRobot1_CtrlDB".sPLCtoROB.User.Cycle.DI261_RingScanReq := FALSE;
            // Action Qualifier=R
            // Token: "KukaRobot1_CtrlDB".sPLCtoROB.User.Cycle.DI262_RingScanComplete
            "KukaRobot1_CtrlDB".sPLCtoROB.User.Cycle.DI262_RingScanComplete := FALSE;
            // Action Qualifier=R
            // Token: "KukaRobot1_CtrlDB".sPLCtoROB.User.Cycle.DI257_TableRingPickReq
            "KukaRobot1_CtrlDB".sPLCtoROB.User.Cycle.DI257_TableRingPickReq := FALSE;
            // Action Qualifier=R
            // Token: "KukaRobot1_CtrlDB".sPLCtoROB.User.Cycle.DI253_ShaftScanPickReq
            "KukaRobot1_CtrlDB".sPLCtoROB.User.Cycle.DI253_ShaftScanPickReq := FALSE;
            // Action Qualifier=R
            // Token: "KukaRobot1_CtrlDB".sPLCtoROB.User.Cycle.DI249_ShaftScanPutReq
            "KukaRobot1_CtrlDB".sPLCtoROB.User.Cycle.DI249_ShaftScanPutReq := FALSE;
            // Action Qualifier=R
            // Token: "KukaRobot1_CtrlDB".sPLCtoROB.User.Cycle.DI241_PickShaftPalletReq
            "KukaRobot1_CtrlDB".sPLCtoROB.User.Cycle.DI241_PickShaftPalletReq := FALSE;
            // Action Qualifier=R
            // Token: "KukaRobot1_CtrlDB".sPLCtoROB.User.Cycle.DI289_GluePutReq
            "KukaRobot1_CtrlDB".sPLCtoROB.User.Cycle.DI289_GluePutReq := FALSE;
            // Action Qualifier=R
            // Token: "KukaRobot1_CtrlDB".sPLCtoROB.User.Cycle.DI297_MaintainRequest
            "KukaRobot1_CtrlDB".sPLCtoROB.User.Cycle.DI297_MaintainRequest := FALSE;
            // Action Qualifier=R
            // Token: "KukaRobot1_CtrlDB".sPLCtoROB.User.Cycle.DI300_HomeRequest
            "KukaRobot1_CtrlDB".sPLCtoROB.User.Cycle.DI300_HomeRequest := FALSE;
            // Action Qualifier=R
            // Token: "KukaRobot1_CtrlDB".sPLCtoROB.User.Cycle.DI305_GripScan
            "KukaRobot1_CtrlDB".sPLCtoROB.User.Cycle.DI305_GripScan := FALSE;
            // Action Qualifier=R
            // Token: "KukaRobot1_CtrlDB".sPLCtoROB.User.Cycle.DI306_ScanPartComplete
            "KukaRobot1_CtrlDB".sPLCtoROB.User.Cycle.DI306_ScanPartComplete := FALSE;
            // Action Qualifier=R
            // Token: "KukaRobot1_CtrlDB".sPLCtoROB.User.Cycle.DI307_ScanPartFinish
            "KukaRobot1_CtrlDB".sPLCtoROB.User.Cycle.DI307_ScanPartFinish := FALSE;
            // Action Qualifier=R
            // Token: #Auto_Run_after_NG_box_closed
            #Auto_Run_after_NG_box_closed := FALSE;

            // Transition to next step: 929
            IF TRUE THEN  // Sequential transition - review XML for actual condition
                #State := STEP_ST10_Flow5_FRobot_1_BrakeTestFinish;
            END_IF;

        // ===========================================
        // STEP 929: BrakeTestFinish
        // ===========================================
        STEP_ST10_Flow5_FRobot_1_BrakeTestFinish:
            // Action Qualifier=R
            // Token: "Robot_DB".Robot_1.BrakeTest_Req
            "Robot_DB".Robot_1.BrakeTest_Req := FALSE;

            // Transition to next step: 373
            IF TRUE THEN  // Sequential transition - review XML for actual condition
                #State := STEP_ST10_Flow5_FRobot_1_StartRobotNG2Put_1;
            END_IF;

        // ===========================================
        // STEP 373: StartRobotNG2Put_1
        // ===========================================
        STEP_ST10_Flow5_FRobot_1_StartRobotNG2Put_1:
            // Action Qualifier=N
            // Token: "KukaRobot1_CtrlDB".sPLCtoROB.User.Cycle.DI266_LoadShaftScanNGReq2
            "KukaRobot1_CtrlDB".sPLCtoROB.User.Cycle.DI266_LoadShaftScanNGReq2;

            // Transition to next step: 319
            IF TRUE THEN  // Sequential transition - review XML for actual condition
                #State := STEP_ST10_Flow5_FRobot_1_WaitPos4ScanFinish;
            END_IF;

        // ===========================================
        // STEP 319: WaitPos4ScanFinish
        // ===========================================
        STEP_ST10_Flow5_FRobot_1_WaitPos4ScanFinish:
            // No actions in XML

            // Transition to next step: 327
            IF TRUE THEN  // Sequential transition - review XML for actual condition
                #State := STEP_ST10_Flow5_FRobot_1_WaitRobotFinish;
            END_IF;

        // ===========================================
        // STEP 327: WaitRobotFinish
        // ===========================================
        STEP_ST10_Flow5_FRobot_1_WaitRobotFinish:
            // No actions in XML

            // Transition to next step: 899
            IF TRUE THEN  // Sequential transition - review XML for actual condition
                #State := STEP_ST10_Flow5_FRobot_1_WaitR1HomePosFinsh_1;
            END_IF;

        // ===========================================
        // STEP 899: WaitR1HomePosFinsh_1
        // ===========================================
        STEP_ST10_Flow5_FRobot_1_WaitR1HomePosFinsh_1:
            // No actions in XML

            // Transition to next step: 165
            IF TRUE THEN  // Sequential transition - review XML for actual condition
                #State := STEP_ST10_Flow5_FRobot_1_NG1Put_2_ShaftScan;
            END_IF;

        // ===========================================
        // STEP 165: NG1Put_2/ShaftScan
        // ===========================================
        STEP_ST10_Flow5_FRobot_1_NG1Put_2_ShaftScan:
            // Action Qualifier=S
            // Token: "AutoProcessControl".Robot_1.NGPutFlag
            "AutoProcessControl".Robot_1.NGPutFlag := TRUE;
            // Action Qualifier=R
            // Token: #ioPM_Inface.ProcessComplete
            #ioPM_Inface.ProcessComplete := FALSE;
            // Action Qualifier=S
            // Token: #ioPM_Inface.ProcessStart
            #ioPM_Inface.ProcessStart := TRUE;

            // Transition to next step: 383
            IF TRUE THEN  // Sequential transition - review XML for actual condition
                #State := STEP_ST10_Flow5_FRobot_1_FlagReset;
            END_IF;

        // ===========================================
        // STEP 383: FlagReset
        // ===========================================
        STEP_ST10_Flow5_FRobot_1_FlagReset:
            // Action Qualifier=R
            // Token: "AutoProcessControl".Robot_1.GluePutFlag
            "AutoProcessControl".Robot_1.GluePutFlag := FALSE;
            // Action Qualifier=R
            // Token: "AutoProcessControl".Robot_1.NGPutFlag
            "AutoProcessControl".Robot_1.NGPutFlag := FALSE;

            // Transition to next step: 599
            IF TRUE THEN  // Sequential transition - review XML for actual condition
                #State := STEP_ST10_Flow5_FRobot_1_PressRingPutProcessFinish;
            END_IF;

        // ===========================================
        // STEP 599: PressRingPutProcessFinish
        // ===========================================
        STEP_ST10_Flow5_FRobot_1_PressRingPutProcessFinish:
            // Action Qualifier=S
            // Token: #ioPM_Inface.ProcessComplete
            #ioPM_Inface.ProcessComplete := TRUE;
            // Action Qualifier=R
            // Token: #ioPM_Inface.ProcessStart
            #ioPM_Inface.ProcessStart := FALSE;

            // Transition to next step: 376
            IF TRUE THEN  // Sequential transition - review XML for actual condition
                #State := STEP_ST10_Flow5_FRobot_1_StartRobotNG3Put;
            END_IF;

        // ===========================================
        // STEP 376: StartRobotNG3Put
        // ===========================================
        STEP_ST10_Flow5_FRobot_1_StartRobotNG3Put:
            // Action Qualifier=N
            // Token: "KukaRobot1_CtrlDB".sPLCtoROB.User.Cycle.DI267_LoadRingScanNGReq3
            "KukaRobot1_CtrlDB".sPLCtoROB.User.Cycle.DI267_LoadRingScanNGReq3;

            // Transition to next step: 246
            IF TRUE THEN  // Sequential transition - review XML for actual condition
                #State := STEP_ST10_Flow5_FRobot_1_ScanStart;
            END_IF;

        // ===========================================
        // STEP 246: ScanStart
        // ===========================================
        STEP_ST10_Flow5_FRobot_1_ScanStart:
            // Action Qualifier=S
            // Token: "KeyenceSR1000Ctrl_804A1DB".ioAutoTrigger
            "KeyenceSR1000Ctrl_804A1DB".ioAutoTrigger := TRUE;

            // Transition to next step: 328
            IF TRUE THEN  // Sequential transition - review XML for actual condition
                #State := STEP_ST10_Flow5_FRobot_1_StartRobotPutBuffer;
            END_IF;

        // ===========================================
        // STEP 328: StartRobotPutBuffer
        // ===========================================
        STEP_ST10_Flow5_FRobot_1_StartRobotPutBuffer:
            // Action Qualifier=N
            // Token: "KukaRobot1_CtrlDB".sPLCtoROB.User.Cycle.DI249_ShaftScanPutReq
            "KukaRobot1_CtrlDB".sPLCtoROB.User.Cycle.DI249_ShaftScanPutReq;

            // Transition to next step: 911
            IF TRUE THEN  // Sequential transition - review XML for actual condition
                #State := STEP_ST10_Flow5_FRobot_1_WaitMasteringTestFinish;
            END_IF;

        // ===========================================
        // STEP 911: WaitMasteringTestFinish
        // ===========================================
        STEP_ST10_Flow5_FRobot_1_WaitMasteringTestFinish:
            // No actions in XML

            // Transition to next step: 381
            IF TRUE THEN  // Sequential transition - review XML for actual condition
                #State := STEP_ST10_Flow5_FRobot_1_WaitRobotStartHome;
            END_IF;

        // ===========================================
        // STEP 381: WaitRobotStartHome
        // ===========================================
        STEP_ST10_Flow5_FRobot_1_WaitRobotStartHome:
            // No actions in XML

            // Transition to next step: 247
            IF TRUE THEN  // Sequential transition - review XML for actual condition
                #State := STEP_ST10_Flow5_FRobot_1_WaitScanCompletely;
            END_IF;

        // ===========================================
        // STEP 247: WaitScanCompletely
        // ===========================================
        STEP_ST10_Flow5_FRobot_1_WaitScanCompletely:
            // No actions in XML

            // Transition to next step: 262
            IF TRUE THEN  // Sequential transition - review XML for actual condition
                #State := STEP_ST10_Flow5_FRobot_1_DataMove_4;
            END_IF;

        // ===========================================
        // STEP 262: DataMove_4
        // ===========================================
        STEP_ST10_Flow5_FRobot_1_DataMove_4:
            // Action Qualifier=N, Event="S1"
            // Token: "AutoProcessData".F_Robot1Grip1 := "AutoProcessData".B_Press1
            "AutoProcessData".F_Robot1Grip1 := "AutoProcessData".B_Press1;
            // Action Qualifier=N, Event="S1"
            // Token: "AutoProcessData".B_Press1 := "AutoProcessData".ClearData
            "AutoProcessData".B_Press1 := "AutoProcessData".ClearData;

            // Transition to next step: 243
            IF TRUE THEN  // Sequential transition - review XML for actual condition
                #State := STEP_ST10_Flow5_FRobot_1_Grip1PartStatus;
            END_IF;

        // ===========================================
        // STEP 243: Grip1PartStatus
        // ===========================================
        STEP_ST10_Flow5_FRobot_1_Grip1PartStatus:
            // Action Qualifier=N
            // Token: "AutoProcessData".F_Robot1Grip1.PartStatus := 100
            "AutoProcessData".F_Robot1Grip1.PartStatus := 100;

            // Transition to next step: 334
            IF TRUE THEN  // Sequential transition - review XML for actual condition
                #State := STEP_ST10_Flow5_FRobot_1_StartRobotScanGripperCode;
            END_IF;

        // ===========================================
        // STEP 334: StartRobotScanGripperCode
        // ===========================================
        STEP_ST10_Flow5_FRobot_1_StartRobotScanGripperCode:
            // Action Qualifier=N
            // Token: "KukaRobot1_CtrlDB".sPLCtoROB.User.Cycle.DI305_GripScan
            "KukaRobot1_CtrlDB".sPLCtoROB.User.Cycle.DI305_GripScan;

            // Transition to next step: 359
            IF TRUE THEN  // Sequential transition - review XML for actual condition
                #State := STEP_ST10_Flow5_FRobot_1_WaitRobotFinish_5;
            END_IF;

        // ===========================================
        // STEP 359: WaitRobotFinish_5
        // ===========================================
        STEP_ST10_Flow5_FRobot_1_WaitRobotFinish_5:
            // No actions in XML

            // Transition to next step: 346
            IF TRUE THEN  // Sequential transition - review XML for actual condition
                #State := STEP_ST10_Flow5_FRobot_1_WaitRobotGripHaveStatus;
            END_IF;

        // ===========================================
        // STEP 346: WaitRobotGripHaveStatus
        // ===========================================
        STEP_ST10_Flow5_FRobot_1_WaitRobotGripHaveStatus:
            // No actions in XML

            // Transition to next step: 343
            IF TRUE THEN  // Sequential transition - review XML for actual condition
                #State := STEP_ST10_Flow5_FRobot_1_WaitRobotFinish_1;
            END_IF;

        // ===========================================
        // STEP 343: WaitRobotFinish_1
        // ===========================================
        STEP_ST10_Flow5_FRobot_1_WaitRobotFinish_1:
            // No actions in XML

            // Transition to next step: 336
            IF TRUE THEN  // Sequential transition - review XML for actual condition
                #State := STEP_ST10_Flow5_FRobot_1_WaitGripperPos1ScanFinish;
            END_IF;

        // ===========================================
        // STEP 336: WaitGripperPos1ScanFinish
        // ===========================================
        STEP_ST10_Flow5_FRobot_1_WaitGripperPos1ScanFinish:
            // No actions in XML

            // Transition to next step: 316
            IF TRUE THEN  // Sequential transition - review XML for actual condition
                #State := STEP_ST10_Flow5_FRobot_1_RobotStart;
            END_IF;

        // ===========================================
        // STEP 316: RobotStart
        // ===========================================
        STEP_ST10_Flow5_FRobot_1_RobotStart:
            // Action Qualifier=N
            // Token: "KukaRobot1_CtrlDB".ioAutoStart
            "KukaRobot1_CtrlDB".ioAutoStart;

            // Transition to next step: 313
            IF TRUE THEN  // Sequential transition - review XML for actual condition
                #State := STEP_ST10_Flow5_FRobot_1_WaitRobotReachPos2;
            END_IF;

        // ===========================================
        // STEP 313: WaitRobotReachPos2
        // ===========================================
        STEP_ST10_Flow5_FRobot_1_WaitRobotReachPos2:
            // No actions in XML

            // Transition to next step: 140
            IF TRUE THEN  // Sequential transition - review XML for actual condition
                #State := STEP_ST10_Flow5_FRobot_1_PressShaftPut;
            END_IF;

        // ===========================================
        // STEP 140: PressShaftPut
        // ===========================================
        STEP_ST10_Flow5_FRobot_1_PressShaftPut:
            // Action Qualifier=R
            // Token: #ioPM_Inface.ProcessComplete
            #ioPM_Inface.ProcessComplete := FALSE;
            // Action Qualifier=S
            // Token: #ioPM_Inface.ProcessStart
            #ioPM_Inface.ProcessStart := TRUE;

            // Transition to next step: 317
            IF TRUE THEN  // Sequential transition - review XML for actual condition
                #State := STEP_ST10_Flow5_FRobot_1_RobotHome;
            END_IF;

        // ===========================================
        // STEP 317: RobotHome
        // ===========================================
        STEP_ST10_Flow5_FRobot_1_RobotHome:
            // Action Qualifier=N
            // Token: "KukaRobot1_CtrlDB".ioSrartHome
            "KukaRobot1_CtrlDB".ioSrartHome;

            // Transition to next step: 342
            IF TRUE THEN  // Sequential transition - review XML for actual condition
                #State := STEP_ST10_Flow5_FRobot_1_WaitGripperPos4ScanFinish;
            END_IF;

        // ===========================================
        // STEP 342: WaitGripperPos4ScanFinish
        // ===========================================
        STEP_ST10_Flow5_FRobot_1_WaitGripperPos4ScanFinish:
            // No actions in XML

            // Transition to next step: 353
            IF TRUE THEN  // Sequential transition - review XML for actual condition
                #State := STEP_ST10_Flow5_FRobot_1_WaitRobotFinish_3;
            END_IF;

        // ===========================================
        // STEP 353: WaitRobotFinish_3
        // ===========================================
        STEP_ST10_Flow5_FRobot_1_WaitRobotFinish_3:
            // No actions in XML

            // Transition to next step: 363
            IF TRUE THEN  // Sequential transition - review XML for actual condition
                #State := STEP_ST10_Flow5_FRobot_1_WaitRobotGripStatus_1;
            END_IF;

        // ===========================================
        // STEP 363: WaitRobotGripStatus_1
        // ===========================================
        STEP_ST10_Flow5_FRobot_1_WaitRobotGripStatus_1:
            // No actions in XML

            // Transition to next step: 312
            IF TRUE THEN  // Sequential transition - review XML for actual condition
                #State := STEP_ST10_Flow5_FRobot_1_WaitPos2ScanFinish;
            END_IF;

        // ===========================================
        // STEP 312: WaitPos2ScanFinish
        // ===========================================
        STEP_ST10_Flow5_FRobot_1_WaitPos2ScanFinish:
            // No actions in XML

            // Transition to next step: 10
            IF TRUE THEN  // Sequential transition - review XML for actual condition
                #State := STEP_ST10_Flow5_FRobot_1_S10_InitialFinish;
            END_IF;

        // ===========================================
        // STEP 10: S10_InitialFinish
        // ===========================================
        STEP_ST10_Flow5_FRobot_1_S10_InitialFinish:
            // Action Qualifier=S
            // Token: #ioPM_Inface.InitialOK
            #ioPM_Inface.InitialOK := TRUE;

            // Transition to next step: 349
            IF TRUE THEN  // Sequential transition - review XML for actual condition
                #State := STEP_ST10_Flow5_FRobot_1_PutBufferFinish_1;
            END_IF;

        // ===========================================
        // STEP 349: PutBufferFinish_1
        // ===========================================
        STEP_ST10_Flow5_FRobot_1_PutBufferFinish_1:
            // Action Qualifier=S
            // Token: #ioPM_Inface.ProcessComplete
            #ioPM_Inface.ProcessComplete := TRUE;
            // Action Qualifier=R
            // Token: #ioPM_Inface.ProcessStart
            #ioPM_Inface.ProcessStart := FALSE;

            // Transition to next step: 362
            IF TRUE THEN  // Sequential transition - review XML for actual condition
                #State := STEP_ST10_Flow5_FRobot_1_WaitRobotFinish_6;
            END_IF;

        // ===========================================
        // STEP 362: WaitRobotFinish_6
        // ===========================================
        STEP_ST10_Flow5_FRobot_1_WaitRobotFinish_6:
            // No actions in XML

            // Transition to next step: 337
            IF TRUE THEN  // Sequential transition - review XML for actual condition
                #State := STEP_ST10_Flow5_FRobot_1_RobotScanGripperReachPos2;
            END_IF;

        // ===========================================
        // STEP 337: RobotScanGripperReachPos2
        // ===========================================
        STEP_ST10_Flow5_FRobot_1_RobotScanGripperReachPos2:
            // No actions in XML

            // Transition to next step: 244
            IF TRUE THEN  // Sequential transition - review XML for actual condition
                #State := STEP_ST10_Flow5_FRobot_1_Grip2PartStatus;
            END_IF;

        // ===========================================
        // STEP 244: Grip2PartStatus
        // ===========================================
        STEP_ST10_Flow5_FRobot_1_Grip2PartStatus:
            // Action Qualifier=N
            // Token: "AutoProcessData".F_Robot1Grip2.PartStatus := 100
            "AutoProcessData".F_Robot1Grip2.PartStatus := 100;

            // Transition to next step: 366
            IF TRUE THEN  // Sequential transition - review XML for actual condition
                #State := STEP_ST10_Flow5_FRobot_1_WaitRobotGripStatus_2;
            END_IF;

        // ===========================================
        // STEP 366: WaitRobotGripStatus_2
        // ===========================================
        STEP_ST10_Flow5_FRobot_1_WaitRobotGripStatus_2:
            // No actions in XML

            // Transition to next step: 322
            IF TRUE THEN  // Sequential transition - review XML for actual condition
                #State := STEP_ST10_Flow5_FRobot_1_WaitRobotReachPos6;
            END_IF;

        // ===========================================
        // STEP 322: WaitRobotReachPos6
        // ===========================================
        STEP_ST10_Flow5_FRobot_1_WaitRobotReachPos6:
            // No actions in XML

            // Transition to next step: 4
            IF TRUE THEN  // Sequential transition - review XML for actual condition
                #State := STEP_ST10_Flow5_FRobot_1_RobotSpeed;
            END_IF;

        // ===========================================
        // STEP 4: RobotSpeed
        // ===========================================
        STEP_ST10_Flow5_FRobot_1_RobotSpeed:
            // Action Qualifier=N
            // Token: "KukaRobot1_CtrlDB".iSpeedValue := 20
            "KukaRobot1_CtrlDB".iSpeedValue := 20;

            // Transition to next step: 900
            IF TRUE THEN  // Sequential transition - review XML for actual condition
                #State := STEP_ST10_Flow5_FRobot_1_RobotTest;
            END_IF;

        // ===========================================
        // STEP 900: RobotTest
        // ===========================================
        STEP_ST10_Flow5_FRobot_1_RobotTest:
            // No actions in XML

            // Transition to next step: 703
            IF TRUE THEN  // Sequential transition - review XML for actual condition
                #State := STEP_ST10_Flow5_FRobot_1_WaitRobotHomeRequest;
            END_IF;

        // ===========================================
        // STEP 703: WaitRobotHomeRequest
        // ===========================================
        STEP_ST10_Flow5_FRobot_1_WaitRobotHomeRequest:
            // Action Qualifier=R
            // Token: "ChangeOver_DB".Robot_1.MaintenancePosReqSelFlag
            "ChangeOver_DB".Robot_1.MaintenancePosReqSelFlag := FALSE;

            // Transition to next step: 120
            IF TRUE THEN  // Sequential transition - review XML for actual condition
                #State := STEP_ST10_Flow5_FRobot_1_PutBuffer;
            END_IF;

        // ===========================================
        // STEP 120: PutBuffer
        // ===========================================
        STEP_ST10_Flow5_FRobot_1_PutBuffer:
            // Action Qualifier=R
            // Token: #ioPM_Inface.ProcessComplete
            #ioPM_Inface.ProcessComplete := FALSE;
            // Action Qualifier=S
            // Token: #ioPM_Inface.ProcessStart
            #ioPM_Inface.ProcessStart := TRUE;

            // Transition to next step: 352
            IF TRUE THEN  // Sequential transition - review XML for actual condition
                #State := STEP_ST10_Flow5_FRobot_1_StartRobotPickTable;
            END_IF;

        // ===========================================
        // STEP 352: StartRobotPickTable
        // ===========================================
        STEP_ST10_Flow5_FRobot_1_StartRobotPickTable:
            // Action Qualifier=N
            // Token: "KukaRobot1_CtrlDB".sPLCtoROB.User.Cycle.DI257_TableRingPickReq
            "KukaRobot1_CtrlDB".sPLCtoROB.User.Cycle.DI257_TableRingPickReq;

            // Transition to next step: 399
            IF TRUE THEN  // Sequential transition - review XML for actual condition
                #State := STEP_ST10_Flow5_FRobot_1_PickBufferFinish;
            END_IF;

        // ===========================================
        // STEP 399: PickBufferFinish
        // ===========================================
        STEP_ST10_Flow5_FRobot_1_PickBufferFinish:
            // Action Qualifier=S
            // Token: #ioPM_Inface.ProcessComplete
            #ioPM_Inface.ProcessComplete := TRUE;
            // Action Qualifier=R
            // Token: #ioPM_Inface.ProcessStart
            #ioPM_Inface.ProcessStart := FALSE;

            // Transition to next step: 339
            IF TRUE THEN  // Sequential transition - review XML for actual condition
                #State := STEP_ST10_Flow5_FRobot_1_RobotScanGripperReachPos3;
            END_IF;

        // ===========================================
        // STEP 339: RobotScanGripperReachPos3
        // ===========================================
        STEP_ST10_Flow5_FRobot_1_RobotScanGripperReachPos3:
            // No actions in XML

            // Transition to next step: 380
            IF TRUE THEN  // Sequential transition - review XML for actual condition
                #State := STEP_ST10_Flow5_FRobot_1_Grip2SensorError;
            END_IF;

        // ===========================================
        // STEP 380: Grip2SensorError
        // ===========================================
        STEP_ST10_Flow5_FRobot_1_Grip2SensorError:
            // No actions in XML

            // Transition to next step: 364
            IF TRUE THEN  // Sequential transition - review XML for actual condition
                #State := STEP_ST10_Flow5_FRobot_1_StartRobotPressPick;
            END_IF;

        // ===========================================
        // STEP 364: StartRobotPressPick
        // ===========================================
        STEP_ST10_Flow5_FRobot_1_StartRobotPressPick:
            // Action Qualifier=N
            // Token: "KukaRobot1_CtrlDB".sPLCtoROB.User.Cycle.DI281_PressPickShaftReq
            "KukaRobot1_CtrlDB".sPLCtoROB.User.Cycle.DI281_PressPickShaftReq;

            // Transition to next step: 450
            IF TRUE THEN  // Sequential transition - review XML for actual condition
                #State := STEP_ST10_Flow5_FRobot_1_ScanRingProcess;
            END_IF;

        // ===========================================
        // STEP 450: ScanRingProcess
        // ===========================================
        STEP_ST10_Flow5_FRobot_1_ScanRingProcess:
            // No actions in XML

            // Transition to next step: 650
            IF TRUE THEN  // Sequential transition - review XML for actual condition
                #State := STEP_ST10_Flow5_FRobot_1_GluePutProcess;
            END_IF;

        // ===========================================
        // STEP 650: GluePutProcess
        // ===========================================
        STEP_ST10_Flow5_FRobot_1_GluePutProcess:
            // No actions in XML

            // Transition to next step: 750
            IF TRUE THEN  // Sequential transition - review XML for actual condition
                #State := STEP_ST10_Flow5_FRobot_1_NG_2_PutProcess;
            END_IF;

        // ===========================================
        // STEP 750: NG 2 PutProcess
        // ===========================================
        STEP_ST10_Flow5_FRobot_1_NG_2_PutProcess:
            // No actions in XML

            // Transition to next step: 370
            IF TRUE THEN  // Sequential transition - review XML for actual condition
                #State := STEP_ST10_Flow5_FRobot_1_StartRobotNGPut;
            END_IF;

        // ===========================================
        // STEP 370: StartRobotNGPut
        // ===========================================
        STEP_ST10_Flow5_FRobot_1_StartRobotNGPut:
            // Action Qualifier=N
            // Token: "KukaRobot1_CtrlDB".sPLCtoROB.User.Cycle.DI265_LoadPressNGReq1
            "KukaRobot1_CtrlDB".sPLCtoROB.User.Cycle.DI265_LoadPressNGReq1;

            // Transition to next step: 258
            IF TRUE THEN  // Sequential transition - review XML for actual condition
                #State := STEP_ST10_Flow5_FRobot_1_Data_Clear_2;
            END_IF;

        // ===========================================
        // STEP 258: Data Clear_2
        // ===========================================
        STEP_ST10_Flow5_FRobot_1_Data_Clear_2:
            // Action Qualifier=N, Event="S1"
            // Token: "AutoProcessData".F_Robot1Grip2 := "AutoProcessData".ClearData
            "AutoProcessData".F_Robot1Grip2 := "AutoProcessData".ClearData;

            // Transition to next step: 252
            IF TRUE THEN  // Sequential transition - review XML for actual condition
                #State := STEP_ST10_Flow5_FRobot_1_DataClear;
            END_IF;

        // ===========================================
        // STEP 252: DataClear
        // ===========================================
        STEP_ST10_Flow5_FRobot_1_DataClear:
            // Action Qualifier=N, Event="S1"
            // Token: "AutoProcessData".F_Robot1Grip1 := "AutoProcessData".ClearData
            "AutoProcessData".F_Robot1Grip1 := "AutoProcessData".ClearData;

            // Transition to next step: 649
            IF TRUE THEN  // Sequential transition - review XML for actual condition
                #State := STEP_ST10_Flow5_FRobot_1_PressPickProcessFinish_;
            END_IF;

        // ===========================================
        // STEP 649: PressPickProcessFinish_
        // ===========================================
        STEP_ST10_Flow5_FRobot_1_PressPickProcessFinish_:
            // Action Qualifier=S
            // Token: #ioPM_Inface.ProcessComplete
            #ioPM_Inface.ProcessComplete := TRUE;
            // Action Qualifier=R
            // Token: #ioPM_Inface.ProcessStart
            #ioPM_Inface.ProcessStart := FALSE;

            // Transition to next step: 125
            IF TRUE THEN  // Sequential transition - review XML for actual condition
                #State := STEP_ST10_Flow5_FRobot_1_PickBuffer;
            END_IF;

        // ===========================================
        // STEP 125: PickBuffer
        // ===========================================
        STEP_ST10_Flow5_FRobot_1_PickBuffer:
            // Action Qualifier=R
            // Token: #ioPM_Inface.ProcessComplete
            #ioPM_Inface.ProcessComplete := FALSE;
            // Action Qualifier=S
            // Token: #ioPM_Inface.ProcessStart
            #ioPM_Inface.ProcessStart := TRUE;

            // Transition to next step: 449
            IF TRUE THEN  // Sequential transition - review XML for actual condition
                #State := STEP_ST10_Flow5_FRobot_1_PickTableProcessFinish;
            END_IF;

        // ===========================================
        // STEP 449: PickTableProcessFinish
        // ===========================================
        STEP_ST10_Flow5_FRobot_1_PickTableProcessFinish:
            // Action Qualifier=S
            // Token: #ioPM_Inface.ProcessComplete
            #ioPM_Inface.ProcessComplete := TRUE;
            // Action Qualifier=R
            // Token: #ioPM_Inface.ProcessStart
            #ioPM_Inface.ProcessStart := FALSE;

            // Transition to next step: 550
            IF TRUE THEN  // Sequential transition - review XML for actual condition
                #State := STEP_ST10_Flow5_FRobot_1_PressRingPutProcess;
            END_IF;

        // ===========================================
        // STEP 550: PressRingPutProcess
        // ===========================================
        STEP_ST10_Flow5_FRobot_1_PressRingPutProcess:
            // No actions in XML

            // Transition to next step: 700
            IF TRUE THEN  // Sequential transition - review XML for actual condition
                #State := STEP_ST10_Flow5_FRobot_1_NG_PutProcess;
            END_IF;

        // ===========================================
        // STEP 700: NG PutProcess
        // ===========================================
        STEP_ST10_Flow5_FRobot_1_NG_PutProcess:
            // No actions in XML

            // Transition to next step: 345
            IF TRUE THEN  // Sequential transition - review XML for actual condition
                #State := STEP_ST10_Flow5_FRobot_1_WaitRobotFinish_2;
            END_IF;

        // ===========================================
        // STEP 345: WaitRobotFinish_2
        // ===========================================
        STEP_ST10_Flow5_FRobot_1_WaitRobotFinish_2:
            // No actions in XML

            // Transition to next step: 145
            IF TRUE THEN  // Sequential transition - review XML for actual condition
                #State := STEP_ST10_Flow5_FRobot_1_PressRingPut;
            END_IF;

        // ===========================================
        // STEP 145: PressRingPut
        // ===========================================
        STEP_ST10_Flow5_FRobot_1_PressRingPut:
            // Action Qualifier=R
            // Token: #ioPM_Inface.ProcessComplete
            #ioPM_Inface.ProcessComplete := FALSE;
            // Action Qualifier=S
            // Token: #ioPM_Inface.ProcessStart
            #ioPM_Inface.ProcessStart := TRUE;

            // Transition to next step: 354
            IF TRUE THEN  // Sequential transition - review XML for actual condition
                #State := STEP_ST10_Flow5_FRobot_1_WaitRobotGripHaveStatus_3;
            END_IF;

        // ===========================================
        // STEP 354: WaitRobotGripHaveStatus_3
        // ===========================================
        STEP_ST10_Flow5_FRobot_1_WaitRobotGripHaveStatus_3:
            // No actions in XML

            // Transition to next step: 400
            IF TRUE THEN  // Sequential transition - review XML for actual condition
                #State := STEP_ST10_Flow5_FRobot_1_PickTableProcess;
            END_IF;

        // ===========================================
        // STEP 400: PickTableProcess
        // ===========================================
        STEP_ST10_Flow5_FRobot_1_PickTableProcess:
            // No actions in XML

            // Transition to next step: 314
            IF TRUE THEN  // Sequential transition - review XML for actual condition
                #State := STEP_ST10_Flow5_FRobot_1_WaitRobotReachPos3;
            END_IF;

        // ===========================================
        // STEP 314: WaitRobotReachPos3
        // ===========================================
        STEP_ST10_Flow5_FRobot_1_WaitRobotReachPos3:
            // No actions in XML

            // Transition to next step: 850
            IF TRUE THEN  // Sequential transition - review XML for actual condition
                #State := STEP_ST10_Flow5_FRobot_1_Maintenance_Pos;
            END_IF;

        // ===========================================
        // STEP 850: Maintenance Pos
        // ===========================================
        STEP_ST10_Flow5_FRobot_1_Maintenance_Pos:
            // No actions in XML

            // Transition to next step: 600
            IF TRUE THEN  // Sequential transition - review XML for actual condition
                #State := STEP_ST10_Flow5_FRobot_1_PressPickProcess;
            END_IF;

        // ===========================================
        // STEP 600: PressPickProcess
        // ===========================================
        STEP_ST10_Flow5_FRobot_1_PressPickProcess:
            // No actions in XML

            // Transition to next step: 269
            IF TRUE THEN  // Sequential transition - review XML for actual condition
                #State := STEP_ST10_Flow5_FRobot_1_Data_Clear_9;
            END_IF;

        // ===========================================
        // STEP 269: Data Clear_9
        // ===========================================
        STEP_ST10_Flow5_FRobot_1_Data_Clear_9:
            // Action Qualifier=N
            // Token: "AutoProcessData".F_Robot1Grip2 := "AutoProcessData".ClearData
            "AutoProcessData".F_Robot1Grip2 := "AutoProcessData".ClearData;

            // Transition to next step: 100
            IF TRUE THEN  // Sequential transition - review XML for actual condition
                #State := STEP_ST10_Flow5_FRobot_1_ProcessStart;
            END_IF;

        // ===========================================
        // STEP 100: ProcessStart
        // ===========================================
        STEP_ST10_Flow5_FRobot_1_ProcessStart:
            // Action Qualifier=R
            // Token: #ioPM_Inface.InitialRun
            #ioPM_Inface.InitialRun := FALSE;
            // Action Qualifier=R
            // Token: #ioPM_Inface.ProcessComplete
            #ioPM_Inface.ProcessComplete := FALSE;
            // Action Qualifier=R
            // Token: #ioPM_Inface.ProcessStart
            #ioPM_Inface.ProcessStart := FALSE;
            // Action Qualifier=S
            // Token: #ioPM_Inface.InitialOK
            #ioPM_Inface.InitialOK := TRUE;
            // Action Qualifier=S
            // Token: #ioPM_Inface.WaitRunning
            #ioPM_Inface.WaitRunning := TRUE;
            // Action Qualifier=N, Event="S1"
            // Token: #ioPM_Inface.ProcessResult := 0
            #ioPM_Inface.ProcessResult := 0;
            // Action Qualifier=R
            // Token: "ST10_GeneralData".FlowControl_Handshake[5].Start
            "ST10_GeneralData".FlowControl_Handshake[5].Start := FALSE;
            // Action Qualifier=R
            // Token: "ST10_GeneralData".FlowControl_Handshake[5].Done
            "ST10_GeneralData".FlowControl_Handshake[5].Done := FALSE;

            // Transition to next step: 338
            IF TRUE THEN  // Sequential transition - review XML for actual condition
                #State := STEP_ST10_Flow5_FRobot_1_WaitGripperPos2ScanFinish;
            END_IF;

        // ===========================================
        // STEP 338: WaitGripperPos2ScanFinish
        // ===========================================
        STEP_ST10_Flow5_FRobot_1_WaitGripperPos2ScanFinish:
            // No actions in XML

            // Transition to next step: 332
            IF TRUE THEN  // Sequential transition - review XML for actual condition
                #State := STEP_ST10_Flow5_FRobot_1_Gripe2StatusAlarm;
            END_IF;

        // ===========================================
        // STEP 332: Gripe2StatusAlarm
        // ===========================================
        STEP_ST10_Flow5_FRobot_1_Gripe2StatusAlarm:
            // Action Qualifier=S
            // Token: "ST10_DeviceError".F.Robot_1.Grip2Error
            "ST10_DeviceError".F.Robot_1.Grip2Error := TRUE;

            // Transition to next step: 910
            IF TRUE THEN  // Sequential transition - review XML for actual condition
                #State := STEP_ST10_Flow5_FRobot_1_MasteringTest_Req;
            END_IF;

        // ===========================================
        // STEP 910: MasteringTest_Req
        // ===========================================
        STEP_ST10_Flow5_FRobot_1_MasteringTest_Req:
            // Action Qualifier=N
            // Token: "KukaRobot1_CtrlDB".sPLCtoROB.User.Cycle.DI321
            "KukaRobot1_CtrlDB".sPLCtoROB.User.Cycle.DI321;
            // Action Qualifier=N
            // Token: "KukaRobot1_CtrlDB".sPLCtoROB.User.Safety.DI450
            "KukaRobot1_CtrlDB".sPLCtoROB.User.Safety.DI450;

            // Transition to next step: 200
            IF TRUE THEN  // Sequential transition - review XML for actual condition
                #State := STEP_ST10_Flow5_FRobot_1_Tablecode_Scan;
            END_IF;

        // ===========================================
        // STEP 200: Tablecode Scan
        // ===========================================
        STEP_ST10_Flow5_FRobot_1_Tablecode_Scan:
            // No actions in XML

            // Transition to next step: 268
            IF TRUE THEN  // Sequential transition - review XML for actual condition
                #State := STEP_ST10_Flow5_FRobot_1_Data_Clear_8;
            END_IF;

        // ===========================================
        // STEP 268: Data Clear_8
        // ===========================================
        STEP_ST10_Flow5_FRobot_1_Data_Clear_8:
            // Action Qualifier=N, Event="S1"
            // Token: "AutoProcessData".F_Robot1Grip1 := "AutoProcessData".ClearData
            "AutoProcessData".F_Robot1Grip1 := "AutoProcessData".ClearData;

            // Transition to next step: 384
            IF TRUE THEN  // Sequential transition - review XML for actual condition
                #State := STEP_ST10_Flow5_FRobot_1_MES_Online__offline_;
            END_IF;

        // ===========================================
        // STEP 384: MES Online  offline?
        // ===========================================
        STEP_ST10_Flow5_FRobot_1_MES_Online__offline_:
            // No actions in XML

            // Transition to next step: 251
            IF TRUE THEN  // Sequential transition - review XML for actual condition
                #State := STEP_ST10_Flow5_FRobot_1_PartNGStatus;
            END_IF;

        // ===========================================
        // STEP 251: PartNGStatus
        // ===========================================
        STEP_ST10_Flow5_FRobot_1_PartNGStatus:
            // Action Qualifier=N
            // Token: "AutoProcessData".F_Robot1Grip2.PartStatus := 150
            "AutoProcessData".F_Robot1Grip2.PartStatus := 150;

            // Transition to next step: 5
            IF TRUE THEN  // Sequential transition - review XML for actual condition
                #State := STEP_ST10_Flow5_FRobot_1_S5_MESInitial;
            END_IF;

        // ===========================================
        // STEP 5: S5_MESInitial
        // ===========================================
        STEP_ST10_Flow5_FRobot_1_S5_MESInitial:
            // No actions in XML

            // Transition to next step: 308
            IF TRUE THEN  // Sequential transition - review XML for actual condition
                #State := STEP_ST10_Flow5_FRobot_1_StartRobotScanFixtureCode;
            END_IF;

        // ===========================================
        // STEP 308: StartRobotScanFixtureCode
        // ===========================================
        STEP_ST10_Flow5_FRobot_1_StartRobotScanFixtureCode:
            // Action Qualifier=N
            // Token: "KukaRobot1_CtrlDB".sPLCtoROB.User.Cycle.DI225_ScanPosReq
            "KukaRobot1_CtrlDB".sPLCtoROB.User.Cycle.DI225_ScanPosReq;

            // Transition to next step: 920
            IF TRUE THEN  // Sequential transition - review XML for actual condition
                #State := STEP_ST10_Flow5_FRobot_1_BrakeTest_Req;
            END_IF;

        // ===========================================
        // STEP 920: BrakeTest_Req
        // ===========================================
        STEP_ST10_Flow5_FRobot_1_BrakeTest_Req:
            // Action Qualifier=N
            // Token: "KukaRobot1_CtrlDB".sPLCtoROB.User.Cycle.DI329
            "KukaRobot1_CtrlDB".sPLCtoROB.User.Cycle.DI329;
            // Action Qualifier=N
            // Token: "KukaRobot1_CtrlDB".sPLCtoROB.User.Safety.DI451
            "KukaRobot1_CtrlDB".sPLCtoROB.User.Safety.DI451;

            // Transition to next step: 320
            IF TRUE THEN  // Sequential transition - review XML for actual condition
                #State := STEP_ST10_Flow5_FRobot_1_WaitPos5ScanFinish;
            END_IF;

        // ===========================================
        // STEP 320: WaitPos5ScanFinish
        // ===========================================
        STEP_ST10_Flow5_FRobot_1_WaitPos5ScanFinish:
            // No actions in XML

            // Transition to next step: 341
            IF TRUE THEN  // Sequential transition - review XML for actual condition
                #State := STEP_ST10_Flow5_FRobot_1_RobotScanGripperReachPos4;
            END_IF;

        // ===========================================
        // STEP 341: RobotScanGripperReachPos4
        // ===========================================
        STEP_ST10_Flow5_FRobot_1_RobotScanGripperReachPos4:
            // No actions in XML

            // Transition to next step: 499
            IF TRUE THEN  // Sequential transition - review XML for actual condition
                #State := STEP_ST10_Flow5_FRobot_1_ScanRingProcessFinish;
            END_IF;

        // ===========================================
        // STEP 499: ScanRingProcessFinish
        // ===========================================
        STEP_ST10_Flow5_FRobot_1_ScanRingProcessFinish:
            // Action Qualifier=S
            // Token: #ioPM_Inface.ProcessComplete
            #ioPM_Inface.ProcessComplete := TRUE;
            // Action Qualifier=R
            // Token: #ioPM_Inface.ProcessStart
            #ioPM_Inface.ProcessStart := FALSE;

            // Transition to next step: 375
            IF TRUE THEN  // Sequential transition - review XML for actual condition
                #State := STEP_ST10_Flow5_FRobot_1_WaitRobotGripStatus_5;
            END_IF;

        // ===========================================
        // STEP 375: WaitRobotGripStatus_5
        // ===========================================
        STEP_ST10_Flow5_FRobot_1_WaitRobotGripStatus_5:
            // No actions in XML

            // Transition to next step: 132
            IF TRUE THEN  // Sequential transition - review XML for actual condition
                #State := STEP_ST10_Flow5_FRobot_1_Masref_test;
            END_IF;

        // ===========================================
        // STEP 132: Masref_test
        // ===========================================
        STEP_ST10_Flow5_FRobot_1_Masref_test:
            // Action Qualifier=R
            // Token: #ioPM_Inface.ProcessComplete
            #ioPM_Inface.ProcessComplete := FALSE;
            // Action Qualifier=S
            // Token: #ioPM_Inface.ProcessStart
            #ioPM_Inface.ProcessStart := TRUE;

            // Transition to next step: 310
            IF TRUE THEN  // Sequential transition - review XML for actual condition
                #State := STEP_ST10_Flow5_FRobot_1_WaitPos1ScanFinish;
            END_IF;

        // ===========================================
        // STEP 310: WaitPos1ScanFinish
        // ===========================================
        STEP_ST10_Flow5_FRobot_1_WaitPos1ScanFinish:
            // No actions in XML

            // Transition to next step: 358
            IF TRUE THEN  // Sequential transition - review XML for actual condition
                #State := STEP_ST10_Flow5_FRobot_1_StartRobotPressShaftPut;
            END_IF;

        // ===========================================
        // STEP 358: StartRobotPressShaftPut
        // ===========================================
        STEP_ST10_Flow5_FRobot_1_StartRobotPressShaftPut:
            // Action Qualifier=N
            // Token: "KukaRobot1_CtrlDB".sPLCtoROB.User.Cycle.DI273_PressShaftPutReq
            "KukaRobot1_CtrlDB".sPLCtoROB.User.Cycle.DI273_PressShaftPutReq;

            // Transition to next step: 344
            IF TRUE THEN  // Sequential transition - review XML for actual condition
                #State := STEP_ST10_Flow5_FRobot_1_StartRobotPickBuffer;
            END_IF;

        // ===========================================
        // STEP 344: StartRobotPickBuffer
        // ===========================================
        STEP_ST10_Flow5_FRobot_1_StartRobotPickBuffer:
            // Action Qualifier=N
            // Token: "KukaRobot1_CtrlDB".sPLCtoROB.User.Cycle.DI253_ShaftScanPickReq
            "KukaRobot1_CtrlDB".sPLCtoROB.User.Cycle.DI253_ShaftScanPickReq;

            // Transition to next step: 500
            IF TRUE THEN  // Sequential transition - review XML for actual condition
                #State := STEP_ST10_Flow5_FRobot_1_PressShaftPutProcess;
            END_IF;

        // ===========================================
        // STEP 500: PressShaftPutProcess
        // ===========================================
        STEP_ST10_Flow5_FRobot_1_PressShaftPutProcess:
            // No actions in XML

            // Transition to next step: 361
            IF TRUE THEN  // Sequential transition - review XML for actual condition
                #State := STEP_ST10_Flow5_FRobot_1_StartRobotPressRingPut;
            END_IF;

        // ===========================================
        // STEP 361: StartRobotPressRingPut
        // ===========================================
        STEP_ST10_Flow5_FRobot_1_StartRobotPressRingPut:
            // Action Qualifier=N
            // Token: "KukaRobot1_CtrlDB".sPLCtoROB.User.Cycle.DI277_PressRingPutReq
            "KukaRobot1_CtrlDB".sPLCtoROB.User.Cycle.DI277_PressRingPutReq;

            // Transition to next step: 170
            IF TRUE THEN  // Sequential transition - review XML for actual condition
                #State := STEP_ST10_Flow5_FRobot_1_NG1Put_3_RingScan;
            END_IF;

        // ===========================================
        // STEP 170: NG1Put_3/RingScan
        // ===========================================
        STEP_ST10_Flow5_FRobot_1_NG1Put_3_RingScan:
            // Action Qualifier=S
            // Token: "AutoProcessControl".Robot_1.NGPutFlag
            "AutoProcessControl".Robot_1.NGPutFlag := TRUE;
            // Action Qualifier=R
            // Token: #ioPM_Inface.ProcessComplete
            #ioPM_Inface.ProcessComplete := FALSE;
            // Action Qualifier=S
            // Token: #ioPM_Inface.ProcessStart
            #ioPM_Inface.ProcessStart := TRUE;

            // Transition to next step: 749
            IF TRUE THEN  // Sequential transition - review XML for actual condition
                #State := STEP_ST10_Flow5_FRobot_1_NG1_PutProcessFinish;
            END_IF;

        // ===========================================
        // STEP 749: NG1 PutProcessFinish
        // ===========================================
        STEP_ST10_Flow5_FRobot_1_NG1_PutProcessFinish:
            // Action Qualifier=S
            // Token: #ioPM_Inface.ProcessComplete
            #ioPM_Inface.ProcessComplete := TRUE;
            // Action Qualifier=R
            // Token: #ioPM_Inface.ProcessStart
            #ioPM_Inface.ProcessStart := FALSE;

            // Transition to next step: 357
            IF TRUE THEN  // Sequential transition - review XML for actual condition
                #State := STEP_ST10_Flow5_FRobot_1_WaitRobotReachScanPos;
            END_IF;

        // ===========================================
        // STEP 357: WaitRobotReachScanPos
        // ===========================================
        STEP_ST10_Flow5_FRobot_1_WaitRobotReachScanPos:
            // No actions in XML

            // Transition to next step: 115
            IF TRUE THEN  // Sequential transition - review XML for actual condition
                #State := STEP_ST10_Flow5_FRobot_1_PickPallet;
            END_IF;

        // ===========================================
        // STEP 115: PickPallet
        // ===========================================
        STEP_ST10_Flow5_FRobot_1_PickPallet:
            // Action Qualifier=R
            // Token: #ioPM_Inface.ProcessComplete
            #ioPM_Inface.ProcessComplete := FALSE;
            // Action Qualifier=S
            // Token: #ioPM_Inface.ProcessStart
            #ioPM_Inface.ProcessStart := TRUE;

            // Transition to next step: 110
            IF TRUE THEN  // Sequential transition - review XML for actual condition
                #State := STEP_ST10_Flow5_FRobot_1_ScanFixtureCode;
            END_IF;

        // ===========================================
        // STEP 110: ScanFixtureCode
        // ===========================================
        STEP_ST10_Flow5_FRobot_1_ScanFixtureCode:
            // Action Qualifier=R
            // Token: #ioPM_Inface.ProcessComplete
            #ioPM_Inface.ProcessComplete := FALSE;
            // Action Qualifier=S
            // Token: #ioPM_Inface.ProcessStart
            #ioPM_Inface.ProcessStart := TRUE;

            // Transition to next step: 300
            IF TRUE THEN  // Sequential transition - review XML for actual condition
                #State := STEP_ST10_Flow5_FRobot_1_PutBufferProcess;
            END_IF;

        // ===========================================
        // STEP 300: PutBufferProcess
        // ===========================================
        STEP_ST10_Flow5_FRobot_1_PutBufferProcess:
            // No actions in XML

            // Transition to next step: 374
            IF TRUE THEN  // Sequential transition - review XML for actual condition
                #State := STEP_ST10_Flow5_FRobot_1_WaitRobotFinish_10;
            END_IF;

        // ===========================================
        // STEP 374: WaitRobotFinish_10
        // ===========================================
        STEP_ST10_Flow5_FRobot_1_WaitRobotFinish_10:
            // No actions in XML

            // Transition to next step: 704
            IF TRUE THEN  // Sequential transition - review XML for actual condition
                #State := STEP_ST10_Flow5_FRobot_1_ReqRobotToHomePos;
            END_IF;

        // ===========================================
        // STEP 704: ReqRobotToHomePos
        // ===========================================
        STEP_ST10_Flow5_FRobot_1_ReqRobotToHomePos:
            // Action Qualifier=N
            // Token: "KukaRobot1_CtrlDB".sPLCtoROB.User.Cycle.DI300_HomeRequest
            "KukaRobot1_CtrlDB".sPLCtoROB.User.Cycle.DI300_HomeRequest;

            // Transition to next step: 255
            IF TRUE THEN  // Sequential transition - review XML for actual condition
                #State := STEP_ST10_Flow5_FRobot_1_DataMove_1;
            END_IF;

        // ===========================================
        // STEP 255: DataMove_1
        // ===========================================
        STEP_ST10_Flow5_FRobot_1_DataMove_1:
            // Action Qualifier=N, Event="S1"
            // Token: "AutoProcessData".F_Robot1Grip1 := "AutoProcessData".A_ScanRotate
            "AutoProcessData".F_Robot1Grip1 := "AutoProcessData".A_ScanRotate;
            // Action Qualifier=N, Event="S1"
            // Token: "AutoProcessData".A_ScanRotate := "AutoProcessData".ClearData
            "AutoProcessData".A_ScanRotate := "AutoProcessData".ClearData;

            // Transition to next step: 131
            IF TRUE THEN  // Sequential transition - review XML for actual condition
                #State := STEP_ST10_Flow5_FRobot_1_Maintenance;
            END_IF;

        // ===========================================
        // STEP 131: Maintenance
        // ===========================================
        STEP_ST10_Flow5_FRobot_1_Maintenance:
            // Action Qualifier=R
            // Token: #ioPM_Inface.ProcessComplete
            #ioPM_Inface.ProcessComplete := FALSE;
            // Action Qualifier=S
            // Token: #ioPM_Inface.ProcessStart
            #ioPM_Inface.ProcessStart := TRUE;

            // Transition to next step: 155
            IF TRUE THEN  // Sequential transition - review XML for actual condition
                #State := STEP_ST10_Flow5_FRobot_1_GluePut;
            END_IF;

        // ===========================================
        // STEP 155: GluePut
        // ===========================================
        STEP_ST10_Flow5_FRobot_1_GluePut:
            // Action Qualifier=S
            // Token: "AutoProcessControl".Robot_1.GluePutFlag
            "AutoProcessControl".Robot_1.GluePutFlag := TRUE;
            // Action Qualifier=R
            // Token: #ioPM_Inface.ProcessComplete
            #ioPM_Inface.ProcessComplete := FALSE;
            // Action Qualifier=S
            // Token: #ioPM_Inface.ProcessStart
            #ioPM_Inface.ProcessStart := TRUE;

            // Transition to next step: 350
            IF TRUE THEN  // Sequential transition - review XML for actual condition
                #State := STEP_ST10_Flow5_FRobot_1_PickBufferProcess;
            END_IF;

        // ===========================================
        // STEP 350: PickBufferProcess
        // ===========================================
        STEP_ST10_Flow5_FRobot_1_PickBufferProcess:
            // No actions in XML

            // Transition to next step: 699
            IF TRUE THEN  // Sequential transition - review XML for actual condition
                #State := STEP_ST10_Flow5_FRobot_1_GluePutProcessFinish;
            END_IF;

        // ===========================================
        // STEP 699: GluePutProcessFinish
        // ===========================================
        STEP_ST10_Flow5_FRobot_1_GluePutProcessFinish:
            // Action Qualifier=S
            // Token: #ioPM_Inface.ProcessComplete
            #ioPM_Inface.ProcessComplete := TRUE;
            // Action Qualifier=R
            // Token: #ioPM_Inface.ProcessStart
            #ioPM_Inface.ProcessStart := FALSE;
            // Action Qualifier=N
            // Token: "Robot_DB".Robot_1.SpeedCount := "Robot_DB".Robot_1.SpeedCount + 1
            "Robot_DB".Robot_1.SpeedCount := "Robot_DB".Robot_1.SpeedCount + 1;

            // Transition to next step: 299
            IF TRUE THEN  // Sequential transition - review XML for actual condition
                #State := STEP_ST10_Flow5_FRobot_1_PickPalletFinish;
            END_IF;

        // ===========================================
        // STEP 299: PickPalletFinish
        // ===========================================
        STEP_ST10_Flow5_FRobot_1_PickPalletFinish:
            // Action Qualifier=S
            // Token: #ioPM_Inface.ProcessComplete
            #ioPM_Inface.ProcessComplete := TRUE;
            // Action Qualifier=R
            // Token: #ioPM_Inface.ProcessStart
            #ioPM_Inface.ProcessStart := FALSE;

            // Transition to next step: 253
            IF TRUE THEN  // Sequential transition - review XML for actual condition
                #State := STEP_ST10_Flow5_FRobot_1_DataMove;
            END_IF;

        // ===========================================
        // STEP 253: DataMove
        // ===========================================
        STEP_ST10_Flow5_FRobot_1_DataMove:
            // Action Qualifier=N, Event="S1"
            // Token: "AutoProcessData".A_ScanRotate := "AutoProcessData".F_Robot1Grip1
            "AutoProcessData".A_ScanRotate := "AutoProcessData".F_Robot1Grip1;
            // Action Qualifier=N, Event="S1"
            // Token: "AutoProcessData".F_Robot1Grip1 := "AutoProcessData".ClearData
            "AutoProcessData".F_Robot1Grip1 := "AutoProcessData".ClearData;

            // Transition to next step: 549
            IF TRUE THEN  // Sequential transition - review XML for actual condition
                #State := STEP_ST10_Flow5_FRobot_1_PressShaftPutProcessFinish;
            END_IF;

